// TwinCAT 3 PLC project Press
// ProgramVersion: 3.1.4024.0
// libraries:
//   Tc2_MC2, * (Beckhoff Automation GmbH)
//   Tc2_MC2_Drive, * (Beckhoff Automation GmbH)
//   Tc2_MC2_FlyingSaw, * (Beckhoff Automation GmbH)
//   Tc2_Standard, * (Beckhoff Automation GmbH)
//   Tc2_System, * (Beckhoff Automation GmbH)
//   Tc2_Utilities, * (Beckhoff Automation GmbH)
//   Tc3_Module, * (Beckhoff Automation GmbH)
// project tree:
//   DUTs/ ST_VisionData.TcDUT
//   GVLs/ GVL_Alarm.TcGVL, GVL_Axis01.TcGVL, GVL_Axis02.TcGVL, GVL_Axis03.TcGVL, GVL_Axis04.TcGVL, GVL_Calibration.TcGVL, GVL_Conv.TcGVL, GVL_Encoder.TcGVL, GVL_HMI.TcGVL, GVL_Main_Step.TcGVL, GVL_Mastering.TcGVL, GVL_Motion_Step.TcGVL, GVL_System.TcGVL, GVL_Vision.TcGVL, GVL_Vision_Step.TcGVL
//   / PlcTask.TcTTO
//   POUs/Alarm/ Alarm_Error.TcPOU, Alarm_Warring.TcPOU
//   POUs/Axis01_R/ Axis01_Alarm.TcPOU, Axis01_Auto.TcPOU, Axis01_Command.TcPOU, Axis01_Interlock_ST.TcPOU, Axis01_Manual.TcPOU, Axis01_Status.TcPOU
//   POUs/Axis02_X/ Axis02_Alarm.TcPOU, Axis02_Auto.TcPOU, Axis02_Command.TcPOU, Axis02_Interlock_ST.TcPOU, Axis02_Manual.TcPOU, Axis02_Status.TcPOU
//   POUs/Axis03_Y/ Axis03_Alarm.TcPOU, Axis03_Auto.TcPOU, Axis03_Command.TcPOU, Axis03_Interlock_ST.TcPOU, Axis03_Manual.TcPOU, Axis03_Status.TcPOU
//   POUs/Axis04_Z/ Axis04_Alarm.TcPOU, Axis04_Auto.TcPOU, Axis04_Command.TcPOU, Axis04_Manual.TcPOU, Axis04_Set_Work_End_Speed.TcPOU, Axis04_Status.TcPOU
//   POUs/Axis05_Encoder/ Axis05_Status.TcPOU
//   POUs/ Conv.TcPOU, FB_HomeBeforeMoveAX8000.TcPOU, FB_CamTrigger.TcPOU, FB_LRealRingQueue.TcPOU, FB_VisionDataQueue.TcPOU, MAIN.TcPOU
//   POUs/System/ HMI.TcPOU, HOME_MOVE.TcPOU, Initial.TcPOU, Login_Timer.TcPOU, System.TcPOU
//   POUs/Vision/ Mastering.TcPOU, Move_Command.TcPOU, Vision_ST.TcPOU
//   POUs/Work/ GOST.TcPOU, Motion_Step_ST.TcPOU

CONFIGURATION Press
    RESOURCE PLC ON TwinCAT3
        TASK PlcTask(INTERVAL := T#1ms, PRIORITY := 1);
        PROGRAM MAIN WITH PlcTask : MAIN;
    END_RESOURCE
END_CONFIGURATION

// ---- DUTs/ST_VisionData.TcDUT
(* 비전 결과 1세트 — 큐 적재 단위. 좌표 + 해당 캠트리거 위치를 한 묶음으로 보존. *)
TYPE ST_VisionData :
STRUCT
    ID                : DINT;    // 비전 인식 ID (vision이 부여, 압입 추적용)
    X                 : LREAL;   // Data_Read_X
    Y                 : LREAL;   // Data_Read_Y
    Rot               : LREAL;   // Data_Read_R (R 은 IL Set/Reset 예약어라 Rot 사용)
    Cam_Trig_Position : LREAL;   // 이 결과의 캠트리거 시점 엔코더 위치(Target X 보정 기준)
END_STRUCT
END_TYPE

// ---- GVLs/GVL_Alarm.TcGVL
{attribute 'qualified_only'}
VAR_GLOBAL
	
 	System_Estop_OK			: BOOL 	;
//E-StopAlarm 장비 정지	
	E_STOP_Total_Alarm		: BOOL	;
	E_STOP_Alarm01			: BOOL	;		//EMO-Switch ON
	E_STOP_Alarm02			: BOOL	;		//Door Open
	E_STOP_Alarm03			: BOOL	;		//가이드 축 알람			
	E_STOP_Alarm04			: BOOL	;		//X 축 인터락 알람
	E_STOP_Alarm05			: BOOL	;		//Y 축 인터락 알람
	E_STOP_Alarm06			: BOOL	;		//Z 축 인터락 알람
	E_STOP_Alarm07			: BOOL	;		//R 축 인터락 알람
	E_STOP_Alarm08			: BOOL	;		//비전 RUN OFF 알람
	E_STOP_Alarm09			: BOOL	;
	E_STOP_Alarm10			: BOOL	;		//Vision 통신 이상
	E_STOP_Alarm11			: BOOL	;
	E_STOP_Alarm12			: BOOL	;
	E_STOP_Alarm13			: BOOL	;
	E_STOP_Alarm14			: BOOL	;
	E_STOP_Alarm15			: BOOL	;
	E_STOP_Alarm16			: BOOL	;
	E_STOP_Alarm17			: BOOL	;
	E_STOP_Alarm18			: BOOL	;
	E_STOP_Alarm19			: BOOL	;
	E_STOP_Alarm20			: BOOL	;
//Display Alarm 알람
	Display_Alarm01			: BOOL	;		
	Display_Alarm02			: BOOL	;
	Display_Alarm03			: BOOL	;
	Display_Alarm04			: BOOL	;
	Display_Alarm05			: BOOL	;
	Display_Alarm06			: BOOL	;
	Display_Alarm07			: BOOL	;
	Display_Alarm08			: BOOL	;
	Display_Alarm09			: BOOL	;
	Display_Alarm10			: BOOL	;		//Vision 측정 NG
	Display_Alarm11			: BOOL	;
	Display_Alarm12			: BOOL	;
	Display_Alarm13			: BOOL	;
	Display_Alarm14			: BOOL	;	
	Display_Alarm15			: BOOL	;
//Axis01 Motor Alarm
	Axis01_Total_Alarm		: BOOL	;		
	Axis01_Alarm01			: BOOL	;		
	Axis01_Alarm02			: BOOL	;
	Axis01_Alarm03			: BOOL	;		
	Axis01_Alarm04			: BOOL	;		
	Axis01_Alarm05			: BOOL	;		
	Axis01_Alarm06			: BOOL	;		
	Axis01_Alarm07			: BOOL	;		
	Axis01_Alarm08			: BOOL	;		
	Axis01_Alarm09			: BOOL	;		
	Axis01_Alarm10			: BOOL	;	
	Axis01_Alarm11			: BOOL	;
	Axis01_Alarm12			: BOOL	;			
//Axis02 Motor Alarm
	Axis02_Total_Alarm		: BOOL	;		
	Axis02_Alarm01			: BOOL	;		
	Axis02_Alarm02			: BOOL	;
	Axis02_Alarm03			: BOOL	;		
	Axis02_Alarm04			: BOOL	;		
	Axis02_Alarm05			: BOOL	;		
	Axis02_Alarm06			: BOOL	;		
	Axis02_Alarm07			: BOOL	;		
	Axis02_Alarm08			: BOOL	;		
	Axis02_Alarm09			: BOOL	;		
	Axis02_Alarm10			: BOOL	;
	Axis02_Alarm11			: BOOL	;
	Axis02_Alarm12			: BOOL	;		
//Axis03 Motor Alarm
	Axis03_Total_Alarm		: BOOL	;		
	Axis03_Alarm01			: BOOL	;		
	Axis03_Alarm02			: BOOL	;
	Axis03_Alarm03			: BOOL	;		
	Axis03_Alarm04			: BOOL	;		
	Axis03_Alarm05			: BOOL	;		
	Axis03_Alarm06			: BOOL	;		
	Axis03_Alarm07			: BOOL	;		
	Axis03_Alarm08			: BOOL	;		
	Axis03_Alarm09			: BOOL	;		
	Axis03_Alarm10			: BOOL	;		
	Axis03_Alarm11			: BOOL	;
	Axis03_Alarm12			: BOOL	;
//Axis04 Motor Alarm
	Axis04_Total_Alarm		: BOOL	;		
	Axis04_Alarm01			: BOOL	;		
	Axis04_Alarm02			: BOOL	;
	Axis04_Alarm03			: BOOL	;		
	Axis04_Alarm04			: BOOL	;		
	Axis04_Alarm05			: BOOL	;		
	Axis04_Alarm06			: BOOL	;		
	Axis04_Alarm07			: BOOL	;		
	Axis04_Alarm08			: BOOL	;		
	Axis04_Alarm09			: BOOL	;		
	Axis04_Alarm10			: BOOL	;		
	Axis04_Alarm11			: BOOL	;
	Axis04_Alarm12			: BOOL	;
END_VAR

// ---- GVLs/GVL_Axis01.TcGVL
{attribute 'qualified_only'}
VAR_GLOBAL
//Motor_Status								
    Real_Position						:	LREAL	;		// 실제 위치					
    Real_Velocity						:	LREAL	;		// 실제 속도					
	Busy	   						 	:	BOOL	;		// 동작중			
    Homed       					    :	BOOL	;		// 홈 완료 여부						
    Error								:	BOOL	;		// 에러 발생 여부						
    ErrorID								:	UDINT	;		// 에러 코드						
	StandStill							:	BOOL	;		// 동작가능(축정지,작업명령없음,알람없음)	
	Error_Stop							:	BOOL	;		// 에러 스탑(MC_Reset으로만 해제 가능)
	Power_ON							:	BOOL	;			
	Stop								:	BOOL	;
	Ready								:	BOOL	;		//	모터 Ready
	Home_OK								:	BOOL	;		//	모터 홈 동작 완료
		
//Interlock
	Interlock							:	BOOL	:=	FALSE	;
//Motor_Bit		
	Moving_Command						:	BOOL	;
//Motor_Manual
	M_Home_ORG							:	BOOL	;
	M_Home_Pos_Move						:	BOOL	;
	M_Wait_Pos_Move						:	BOOL	;
	M_Target_Pos_Move					:	BOOL	;
	M_Work_End_Pos_Move					:	BOOL	;
	M_Maint_Pos_Move					:	BOOL	;
	M_Tool_Change_Pos_Move				:	BOOL	;
	M_Calibration_Pos_Move				:	BOOL	;
//Motor_Auto
	A_Home_Pos_Move						:	BOOL	;
	A_Wait_Pos_Move						:	BOOL	;
	A_Target_Pos_Move					:	BOOL	;
	A_Work_End_Pos_Move					:	BOOL	;
	A_Maint_Pos_Move					:	BOOL	;
	A_Tool_Change_Pos_Move				:	BOOL	;
	A_Calibration_Pos_Move				:	BOOL	;
	
//Interlock
	Home_ORG_Interlock					:	BOOL	;
	Home_Pos_Interlock					:	BOOL	;
	Wait_Pos_Interlock					:	BOOL	;
	Target_Pos_Interlock				:	BOOL	;
	Work_End_Pos_Interlock				:	BOOL	;
	Maint_Pos_Interlock					:	BOOL	;
	Tool_Change_Pos_Interlock			:	BOOL	;
	Calibration_Pos_Interlock			:	BOOL	;	
	
	
//Motor_Sensor								
	Home_Sensor  		AT%I*	 		:	 BOOL	;				
	CW_Sensor   		AT%I*			:	 BOOL	;		//Motor +Limit		
	CCW_Sensor  		AT%I*			:	 BOOL	;		//Motor -Limit	
		
//Motor_Position								
	Home_Position						:   BOOL	;						
	Wait_Position						:   BOOL	;						
	Target_Position						:   BOOL	;											
	Work_End_Position					:   BOOL	;
	Maint_Position						:	BOOL	;
	Tool_Change_Position				:	BOOL	;
	Calibration_Position				:	BOOL	;		

//HMI
	HMI_Home_PB							:	BOOL	;
	HMI_Home_Pos_Move_PB				:	BOOL	;
	HMI_Wait_Pos_Move_PB				:	BOOL	;
	HMI_Target_Pos_Move_PB				:	BOOL	;
	HMI_Work_End_Pos_Move_PB			:	BOOL	;
	HMI_Maint_Pos_Move_PB				:	BOOL	;
	HMI_Tool_Change_Move_PB				:	BOOL	;
	HMI_Calibration_Move_PB				:	BOOL	;
	Jog_Forward_PB						:	BOOL	;
	Jog_Backward_PB						:	BOOL	;
	Stop_PB								:	BOOL	;
// Digital Input // P Limit, N Limit
	Digital_Input AT%I*					:	UDINT	;
	
Maint_Position_Data: LREAL;	Power_ON_Delay: BOOL;
	Test_Power_ON: BOOL;
END_VAR
VAR_GLOBAL PERSISTENT
//Motor_Position_Data								
	Home_Position_Data					: 	LREAL	;					
	Wait_Position_Data					: 	LREAL	;					
	Target_Position_Data				: 	LREAL	;							
	Work_End_Position_Data				:	LREAL	;	
	
	Tool_Change_Position_Data			:	LREAL	;
	Calibration_Position_Data			:	LREAL	;
//Motor_Speed_Data
	Work_Speed							:	LREAL	;
	Jog_Speed							:	LREAL	;

END_VAR

VAR_GLOBAL CONSTANT
	Tool_Change_Speed					: 	LREAL := 20 ;
	Calibration_Speed					:	LREAL := 20	;
END_VAR

// ---- GVLs/GVL_Axis02.TcGVL
{attribute 'qualified_only'}
VAR_GLOBAL
//Motor_Status								
    Real_Position						:	LREAL	;		// 실제 위치					
    Real_Velocity						:	LREAL	;		// 실제 속도					
	Busy	   						 	:	BOOL	;		// 동작중			
    Homed       					    :	BOOL	;		// 홈 완료 여부						
    Error								:	BOOL	;		// 에러 발생 여부						
    ErrorID								:	UDINT	;		// 에러 코드						
	StandStill							:	BOOL	;		// 동작가능(축정지,작업명령없음,알람없음)	
	Error_Stop							:	BOOL	;		// 에러 스탑(MC_Reset으로만 해제 가능)
	Power_ON							:	BOOL	;			
	Stop								:	BOOL	;
	Ready								:	BOOL	;		//	모터 Ready
	Home_OK								:	BOOL	;		//	모터 홈 동작 완료
	Work_Offset							:	LREAL	;
	Work_Offset_Move					:	BOOL	;
	Offset_Acceleration					:	LREAL	;
	Accel_Offset						:	LREAL	;
	Speed_Offset						:	LREAL	;
//Interlock
	Interlock							:	BOOL	:=	FALSE	;
//Motor_Bit
	Moving_Command						:	BOOL	;
//Motor_Manual
	M_Home_ORG							:	BOOL	;
	M_Home_Pos_Move						:	BOOL	;
	M_Wait_Pos_Move						:	BOOL	;
	M_Target_Pos_Move					:	BOOL	;
	M_Work_End_Pos_Move					:	BOOL	;
	M_Maint_Pos_Move					:	BOOL	;
	M_Tool_Change_Pos_Move				:	BOOL	;
	M_Calibration_Pos_Move				:	BOOL	;
//Motor_Auto
	A_Home_Pos_Move						:	BOOL	;
	A_Wait_Pos_Move						:	BOOL	;
	A_Target_Pos_Move					:	BOOL	;
	A_Work_End_Pos_Move					:	BOOL	;
	A_Maint_Pos_Move					:	BOOL	;
	A_Tool_Change_Pos_Move				:	BOOL	;
	A_Calibration_Pos_Move				:	BOOL	;
//Interlock
	Home_ORG_Interlock					:	BOOL	;
	Home_Pos_Interlock					:	BOOL	;
	Wait_Pos_Interlock					:	BOOL	;
	Target_Pos_Interlock				:	BOOL	;
	Work_End_Pos_Interlock				:	BOOL	;
	Maint_Pos_Interlock					:	BOOL	;
	Tool_Change_Pos_Interlock			:	BOOL	;
	Calibration_Pos_Interlock			:	BOOL	;
//Motor_Sensor								
	Home_Sensor  		AT%I*	 		:	BOOL	;				
	CW_Sensor   		AT%I*			:	BOOL	;		//Motor +Limit		
	CCW_Sensor  		AT%I*			:	BOOL	;		//Motor -Limit	
		
//Motor_Position								
	Home_Position						:   BOOL	;						
	Wait_Position						:   BOOL	;						
	Target_Position						:   BOOL	;											
	Work_End_Position					:   BOOL	;
	Maint_Position						:	BOOL	;
	Tool_Change_Position				: 	BOOL	;			
	Calibration_Position				: 	BOOL 	;
//HMI
	HMI_Home_PB							:	BOOL	;
	HMI_Home_Pos_Move_PB				:	BOOL	;
	HMI_Wait_Pos_Move_PB				:	BOOL	;
	HMI_Target_Pos_Move_PB				:	BOOL	;
	HMI_Work_End_Pos_Move_PB			:	BOOL	;
	HMI_Maint_Pos_Move_PB				:	BOOL	;
	HMI_Tool_Change_Pos_Move_PB			:	BOOL	;
	HMI_Calibration_Pos_Move_PB			:	BOOL	;
	Jog_Forward_PB						:	BOOL	;
	Jog_Backward_PB						:	BOOL	;
	Stop_PB								:	BOOL	;
//Work_Comp	
	Work_End_Comp						:	BOOL	;
	Home_Comp							:	BOOL	;
// Digital Input // P Limit, N Limit
	Digital_Input AT%I*					: 	UDINT	;




	Power_ON_Delay: BOOL;
	Test_Power_ON: BOOL;
	
END_VAR
VAR_GLOBAL PERSISTENT
//Motor_Position_Data								
	Home_Position_Data					: 	LREAL	;					
	Wait_Position_Data					: 	LREAL	;					
	Target_Position_Data				: 	LREAL	;							
	Work_End_Position_Data				:	LREAL	;
	Maint_Position_Data					:	LREAL	;
	Tool_Change_Position_Data			:	LREAL	;
	Calibration_Position_Data			:	LREAL	;
//Motor_Speed_Data
	Work_Speed							:	LREAL	;
	

END_VAR

VAR_GLOBAL CONSTANT
	Tool_Change_Speed					: 	LREAL := 20 ;
	Calibration_Speed					:	LREAL := 20	;
	Sync_Data							:	LREAL := 20 ;
	Jog_Speed							:	LREAL := 20	;
END_VAR

// ---- GVLs/GVL_Axis03.TcGVL
{attribute 'qualified_only'}
VAR_GLOBAL
//Motor_Status								
    Real_Position						:	LREAL	;		// 실제 위치					
    Real_Velocity						:	LREAL	;		// 실제 속도					
	Busy	   						 	:	BOOL	;		// 동작중			
    Homed       					    :	BOOL	;		// 홈 완료 여부						
    Error								:	BOOL	;		// 에러 발생 여부						
    ErrorID								:	UDINT	;		// 에러 코드						
	StandStill							:	BOOL	;		// 동작가능(축정지,작업명령없음,알람없음)	
	Error_Stop							:	BOOL	;		// 에러 스탑(MC_Reset으로만 해제 가능)
	Power_ON							:	BOOL	;			
	Stop								:	BOOL	;
	Ready								:	BOOL	;		//	모터 Ready
	Home_OK								:	BOOL	;		//	모터 홈 동작 완료

//Interlock
	Interlock							:	BOOL	:=	FALSE	;
//Motor_Bit
	Moving_Command						:	BOOL	;
//Motor_Manual
	M_Home_ORG							:	BOOL	;
	M_Home_Pos_Move						:	BOOL	;
	M_Wait_Pos_Move						:	BOOL	;
	M_Target_Pos_Move					:	BOOL	;
	M_Work_End_Pos_Move					:	BOOL	;
	M_Maint_Pos_Move					:	BOOL	;
	M_Tool_Change_Pos_Move				:	BOOL	;
	M_Calibration_Pos_Move				:	BOOL	;
//Motor_Auto
	A_Home_Pos_Move						:	BOOL	;
	A_Wait_Pos_Move						:	BOOL	;
	A_Target_Pos_Move					:	BOOL	;
	A_Work_End_Pos_Move					:	BOOL	;
	A_Maint_Pos_Move					:	BOOL	;
	A_Tool_Change_Pos_Move				:	BOOL	;
	A_Calibration_Pos_Move				:	BOOL	;
//Interlock
	Home_ORG_Interlock					:	BOOL	;
	Home_Pos_Interlock					:	BOOL	;
	Wait_Pos_Interlock					:	BOOL	;
	Target_Pos_Interlock				:	BOOL	;
	Work_End_Pos_Interlock				:	BOOL	;
	Maint_Pos_Interlock					:	BOOL	;
	Tool_Change_Pos_Interlock			:	BOOL	;
	Calibration_Pos_Interlock			:	BOOL	;

	
//Motor_Sensor								
	Home_Sensor  		AT%I*	 		:	 BOOL	;				
	CW_Sensor   		AT%I*			:	 BOOL	;		//Motor +Limit		
	CCW_Sensor  		AT%I*			:	 BOOL	;		//Motor -Limit	
	
//Motor_Position								
	Home_Position						:   BOOL	;						
	Wait_Position						:   BOOL	;						
	Target_Position						:   BOOL	;											
	Work_End_Position					:   BOOL	;
	Maint_Position						:	BOOL	;
	Tool_Change_Position				:	BOOL	;	
	Calibration_Position				: 	BOOL	;
//HMI
	HMI_Home_PB							:	BOOL	;
	HMI_Home_Pos_Move_PB				:	BOOL	;
	HMI_Wait_Pos_Move_PB				:	BOOL	;
	HMI_Target_Pos_Move_PB				:	BOOL	;
	HMI_Work_End_Pos_Move_PB			:	BOOL	;
	HMI_Maint_Pos_Move_PB				:	BOOL	;
	HMI_Tool_Change_Pos_Move_PB			:	BOOL	;
	HMI_Calibration_Pos_Move_PB			:	BOOL	;
	Jog_Forward_PB						:	BOOL	;
	Jog_Backward_PB						:	BOOL	;
	Stop_PB								:	BOOL	;
	
// Digital Input // P Limit, N Limit
	Digital_Input AT%I*					:	UDINT	;

	Power_ON_Delay: BOOL;
	Test_Power_ON: BOOL;
END_VAR
VAR_GLOBAL PERSISTENT
//Motor_Position_Data								
	Home_Position_Data					: 	LREAL	;					
	Wait_Position_Data					: 	LREAL	;					
	Target_Position_Data				: 	LREAL	;							
	Work_End_Position_Data				:	LREAL	;		
	Maint_Position_Data					:	LREAL	;
	Tool_Change_Position_Data			:	LREAL	;
	Calibration_Position_Data			:	LREAL	;
//Motor_Speed_Data
	Work_Speed							:	LREAL	;
	Jog_Speed							:	LREAL	;
	
END_VAR

VAR_GLOBAL CONSTANT
	Calibration_Speed					: 	LREAL	:= 20;
	Tool_Change_Speed					: 	LREAL	:= 20;
END_VAR

// ---- GVLs/GVL_Axis04.TcGVL
{attribute 'qualified_only'}
VAR_GLOBAL
//Motor_Status								
    Real_Position						:	LREAL	;		// 실제 위치					
    Real_Velocity						:	LREAL	;		// 실제 속도					
	Busy	   						 	:	BOOL	;		// 동작중			
    Homed       					    :	BOOL	;		// 홈 완료 여부						
    Error								:	BOOL	;		// 에러 발생 여부						
    ErrorID								:	UDINT	;		// 에러 코드						
	StandStill							:	BOOL	;		// 동작가능(축정지,작업명령없음,알람없음)	
	Error_Stop							:	BOOL	;		// 에러 스탑(MC_Reset으로만 해제 가능)
	Power_ON							:	BOOL	;			
	Stop								:	BOOL	;
	Ready								:	BOOL	;		//	모터 Ready
	Home_OK								:	BOOL	;		//	모터 홈 동작 완료
	
//Interlock
	Interlock							:	BOOL	:=	FALSE	;
//Motor_Bit
	Moving_Command						:	BOOL	;
M_Home_ORG: BOOL;
	M_Home_Pos_Move						:	BOOL	;
	M_Wait_Pos_Move						:	BOOL	;
	M_Target_Pos_Move					:	BOOL	;
	M_Work_End_Pos_Move					:	BOOL	;
	M_Maint_Pos_Move					:	BOOL	;
	M_Tool_Change_Pos_Move				:	BOOL	;
	M_Calibration_Pos_Move				:	BOOL	;
//Motor_Auto
	A_Home_Pos_Move						:	BOOL	;
	A_Wait_Pos_Move						:	BOOL	;
	A_Target_Pos_Move					:	BOOL	;
	A_Work_End_Pos_Move					:	BOOL	;
	A_Maint_Pos_Move					:	BOOL	;
	A_Tool_Change_Pos_Move				:	BOOL	;
	A_Calibration_Pos_Move				:	BOOL	;
//Interlock
	Home_ORG_Interlock					:	BOOL	;
	Home_Pos_Interlock					:	BOOL	;
	Wait_Pos_Interlock					:	BOOL	;
	Target_Pos_Interlock				:	BOOL	;
	Work_End_Pos_Interlock				:	BOOL	;
	Maint_Pos_Interlock					:	BOOL	;
	Tool_Change_Pos_Interlock			:	BOOL	;
	Calibration_Pos_Interlock			:	BOOL	;
	
//Motor_Sensor								
	Home_Sensor  		AT%I*		 	:	 BOOL	;				
	CW_Sensor   		AT%I*			:	 BOOL	;		//Motor +Limit		
	CCW_Sensor  		AT%I*			:	 BOOL	;		//Motor -Limit	
		
//Motor_Position								
	Home_Position						:   BOOL	;						
	Wait_Position						:   BOOL	;						
	Target_Position						:   BOOL	;											
	Work_End_Position					:   BOOL	;
	Maint_Position						:	BOOL	;
	Tool_Change_Position				:	BOOL	;
	Calibration_Position				:	BOOL	;			

//HMI
	HMI_Home_PB							:	BOOL	;
	HMI_Home_Pos_Move_PB				:	BOOL	;
	HMI_Wait_Pos_Move_PB				:	BOOL	;
	HMI_Target_Pos_Move_PB				:	BOOL	;
	HMI_Work_End_Pos_Move_PB			:	BOOL	;
	HMI_Maint_Pos_Move_PB				:	BOOL	;
	HMI_Tool_Change_Pos_Move_PB			:	BOOL	;
	HMI_Calibration_Pos_Move_PB			:	BOOL	;
	Jog_Forward_PB						:	BOOL	;
	Jog_Backward_PB						:	BOOL	;
	Stop_PB								:	BOOL	;	

// Digital Input // P Limit, N Limit
	Digital_Input AT%I*					: 	UDINT	;	


	Power_ON_Delay: BOOL;
	Test_Power_ON: BOOL;
	
	M_Cleaning_Move: BOOL;
	Cleaning_Move_Position: BOOL;
	M_Mastering_Pos_Move: BOOL;
	Mastering_Position: BOOL;
END_VAR
VAR_GLOBAL PERSISTENT
//Motor_Position_Data								
	Home_Position_Data					: 	LREAL	;					
	Wait_Position_Data					: 	LREAL	;					
	Target_Position_Data				: 	LREAL	;							
	Work_End_Position_Data				:	LREAL	;	
	Maint_Position_Data					:	LREAL	;
	Tool_Change_Position_Data			:	LREAL	;
	Calibration_Position_Data			:	LREAL	;	
	Cleaning_Move_Data: LREAL := 0;
//Motor_Speed_Data
	Work_Speed							:	LREAL	;
	Jog_Speed							:	LREAL	;

//Motor_Torque_Data
	Torque_UP_Limit				AT%Q*	:	UINT	;
	Torque_Down_Limit			AT%Q*	:	UINT	;
	Wait_Speed							: 	LREAL	;
END_VAR

VAR_GLOBAL CONSTANT
	Calibration_Speed					: 	LREAL	:= 20;
	Tool_Change_Speed					: 	LREAL	:= 20;
END_VAR

// ---- GVLs/GVL_Calibration.TcGVL
{attribute 'qualified_only'}
VAR_GLOBAL
	Calibration_Pos_Moving			: 	BOOL	;
	HMI_Calibration_Pos_Move_PB		: 	BOOL	;
	Calibration_comp				: 	BOOL	;
	Calibration_OK					: 	BOOL	;
	All_Motor_Wait_Pos_Moving		: 	BOOL	;
	Calibration_Pos_Interlock 		: 	BOOL	;
	Data_Read_Comp					: 	BOOL	;
	Axis01_Data_Apply_Comp			: 	BOOL	;
	Axis02_Data_Apply_Comp			: 	BOOL	;
	Axis03_Data_Apply_Comp			: 	BOOL	;
	Axis04_Data_Apply_Comp			:   BOOL;
	Motor_Move : BOOL := FALSE;
	
END_VAR

// ---- GVLs/GVL_Conv.TcGVL
{attribute 'qualified_only'}
VAR_GLOBAL
	
	Auto_Mode					AT%I*	:	BOOL	;	// 컨베이어 자동 스위치
	E_STOP						AT%I*	:	BOOL	;	// 컨베이어 E_STOP


	//Output Card 01
	Conv_Motor_CW				AT%Q*	:	BOOL	;	// 컨베이어 전진
	Conv_Motor_CCW				AT%Q*	:	BOOL	;	// 컨베이어 후진
	Conv_Motor_High_Speed		AT%Q*	:	BOOL	;	// 컨베이어 고속
	Conv_Motor_Normal_Speed		AT%Q*	:	BOOL	;	// 컨베이어 중속
	Conv_Motor_Low_Speed		AT%Q*	:	BOOL	;	// 컨베이어 저속

	HMI_Motor_CW						:	BOOL	;	// HMI 컨베이어 전진
	HMI_Motor_CCW						:	BOOL	;	// HMI 컨베이어 후진 
	HMI_Motor_High_Speed				:	BOOL	;	// HMI 컨베이어 고속
	HMI_Motor_Normal_Speed				:	BOOL	;	// HMI 컨베이어 중속
	HMI_Motor_Low_Speed					:	BOOL	;	// HMI 컨베이어 저속
	
	Motor_STOP							:	BOOL	;


	

	

END_VAR

// ---- GVLs/GVL_Encoder.TcGVL
{attribute 'qualified_only'}
VAR_GLOBAL
	Enc_Axis: AXIS_REF;
	Conveyor_Speed :	LREAL	;
	Encoder_Value	:	LREAL	;
	Real_Position: LREAL;
	Real_Velocity: LREAL;
	Count	AT%I*	:INT;
	Conveyor_CW AT%Q* : BOOL	;
	Conveyor_CCW AT%Q* : BOOL	;
	
END_VAR

// ---- GVLs/GVL_HMI.TcGVL
{attribute 'qualified_only'}
VAR_GLOBAL

// HMI Screen NO
    NowScreen_NO            :    INT    ;       // 현재 화면 위치 NO
	ChangeScreen_NO         :    INT    ;       // PLC 요구 화면 NO

	
// HMI 화면 전환	
	AXIS01					:	BOOL	;
	AXIS02					:	BOOL	;
	AXIS03					:	BOOL	;
	AXIS04					:	BOOL	;
	
	AXIS01_LAMP				:	BOOL	;
	AXIS02_LAMP				:	BOOL	;
	AXIS03_LAMP				:	BOOL	;
	AXIS04_LAMP				:	BOOL	;
END_VAR

// ---- GVLs/GVL_Main_Step.TcGVL
{attribute 'qualified_only'}
VAR_GLOBAL
	Status						:	BOOL	;
	NO							:	INT		;
	Wait_Vision					: 	BOOL	;
	Data_Copy					:	BOOL	;
	Vision_Data_Apply			: 	BOOL	;
	Wait_Start_Sensor			: 	BOOL	;
	Moving_Start				: 	BOOL	;
	Axis04_Comp					: 	BOOL	;
	Axis04_Work_Comp			: 	BOOL	;
	Axis04_Work_Comp_Wait		: 	BOOL	;
	Press_5ms					: 	BOOL	;
	Press_Stop					:	BOOL	;
	Axis04_Wait_Pos_Moving		: 	BOOL	;
	Axis02_Work_Comp_Wait		: 	BOOL	;
	Axis02_Wait_Pos_Moving		: 	BOOL	;
	All_Motor_Wait_Pos_Moving	:	BOOL	;
	Vision_Data_Reset			:	BOOL	;
	Vision_Data_Initial			:	BOOL	;
	All_Initial					:	BOOL	;
	Target_Position_Moving		:	BOOL	;
	Press_Start					:	BOOL	;
	Press_Wait					:	BOOL	;
	Axis04_Work_move			:	BOOL	;
	

	Data_Copy_Comp				:	BOOL	;
END_VAR

// ---- GVLs/GVL_Mastering.TcGVL
{attribute 'qualified_only'}
VAR_GLOBAL
	Case_Length_Check_Start 	: 	BOOL;
	Case_Length					:	LREAL;
	mastering_vision_x			:	LREAL;
	Back_Shot_Position			:	LREAL;
	Reshot_Position				:	LREAL;
	Back_Trig					: 	BOOL;
END_VAR

// ---- GVLs/GVL_Motion_Step.TcGVL
{attribute 'qualified_only'}
VAR_GLOBAL
	Status: BOOL;
	No: INT;
	Target_Pos_Moving: BOOL;
	Motion_Start: BOOL;
	Axis02_Work_Wait: BOOL;
	Press_Start: BOOL;
	Axis04_Torque_Controll: BOOL;
	Axis04_Wait_Pos_Moving: BOOL;
	All_Axis_Wait_Pos_Moving: BOOL;
	Work_Comp_Target_Pos_Moving: BOOL;
	All_Initial: BOOL;
	Axis02_Stop: BOOL;
	Z_Press_Start: BOOL;
	Force_Gear_Out: BOOL;   // 실패 abort 시 X축 gear-out 강제 (→ Axis02_Command MC_GearOut.Execute OR 입력)
END_VAR

// ---- GVLs/GVL_System.TcGVL
{attribute 'qualified_only'}
VAR_GLOBAL
// Glovel Bit
	Pulse_100ms					:	BOOL	;			//0.1s Bit
	Pulse_1S					:	BOOL	;			//1S Bit		
// System Bit
	Manual_Mode					:	BOOL	;			//HMI 메뉴얼 모드
	Auto_Mode					:	BOOL	;			//HMI 오토모드
	Stop						:	BOOL	;			//HMI Stop
	Safety_ALL_OK				:	BOOL	;			//EMO+Door
	Test_Mode					:	BOOL	;
	All_Initial					:	BOOL	;
	ToggleBit					:	BOOL	;
	Door_Bypass		AT%Q*		:	BOOL	;			//도어 인터록 바이패스 릴레이 출력 (EL2809 Ch11)
//EMO SW	
	EMO_SWitch		AT%I*		:	BOOL	;

//Fiber Sensor
	Fiber_Sensor	AT%I*	:	BOOL	;

//System_Door_Sensor
	Door_Open		AT%I*		:	BOOL	;

//TowerLamp
	Tower_Lamp_Green	AT%Q*	:	BOOL	;
	Tower_Lamp_Yellow	AT%Q*	:	BOOL	;
	Tower_Lamp_Red		AT%Q*	:	BOOL	;
	Buzzer				AT%Q*	:	BOOL	;
//HMI
	Buzzer_Stop						AT%I*	:	BOOL	;
	Alarm_Reset						AT%I*	:	BOOL	;
//Panel
	DC01_SMPS_OK					AT%I*	:	BOOL	;
	DC02_SMPS_OK					AT%I*	:	BOOL	;
	DC03_SMPS_OK					AT%I*	:	BOOL	;
	Servo_Drive_Control_DC_Power	AT%I*	:	BOOL	;
	Inverter_Power_OK					AT%I*	:	BOOL	;
	Inverter_MC_OK					AT%I*	:	BOOL	;
	MC_OK							AT%I*	:	BOOL	;
	CAM_TRIGGER_FAIL				AT%I*	:	BOOL	;
	Main_Lamp_ON					AT%I*	:	BOOL	;
	PC_Power_CP						AT%I*	:	BOOL	;
	CAM_Lamp_CP						AT%I*	:	BOOL	;
	Ps01_Power_OK					AT%I*	:	BOOL	;
	HMI_Power_OK					AT%I*	:	BOOL	;
	Cam_Power_OK					AT%I*	:	BOOL	;
	Inverter_Alarm_ON					AT%I*	:	BOOL	;
	
	
//Bool
	HMI_Auto_Mode				:	BOOL	;		//HMI 오토모드
	ALL_Motor_Homed				:	BOOL	;		//전체 모터 홈 OK
	ALL_Motor_Home_Position		:	BOOL	;		//전체 모터 홈포지션
	HMI_Manual_Mode				:	BOOL	;		//HMI 메뉴얼 모드
	ALL_Motor_Busy				:	BOOL	;		//전체 모터 동작중
	ALL_Motor_StandStill		:	BOOL	;		//전체 모터 동작 가능
	Moving_Motor_Wait_Position	:	BOOL	;		//X,Y,Z,R Wait Position
	Each_Motor_Homed			:	BOOL	;		//개별 로못 홈
	Each_Motor_Busy				:	BOOL	;		//개별 로봇 동작중
	All_Motor_Stop				:	BOOL	;	
	
	
	
	Test_Data_Read_Comp			: 	BOOL	;
	Test_Continues				: 	BOOL	;
	Calibration_Mode			: 	BOOL	;
	Tool_Change_Mode			: 	BOOL	;
	Tool_Change_Move_PB			: 	BOOL	;	
//홈동작 
	ALL_Wait_Position			: 	BOOL	;
	ALL_Home_Move_PB			:	BOOL	;
	ALL_Home_Move_Start			:	BOOL	;
	Axis01_Home_Move			: 	BOOL	;
	Axis02_Home_Move			: 	BOOL	;
	Axis03_Home_Move			: 	BOOL	;
	Axis04_Home_Move			: 	BOOL	;
	
	Axis01_Home_Pos_Move		: 	BOOL	;
	Axis04_Wait_Pos_Move		:	BOOL	;
	Axis03_Wait_Pos_Move		: 	BOOL	;
	Axis01_Wait_Pos_Move		: 	BOOL	;
	Axis02_Wait_Pos_Move		: 	BOOL	;
	Calibration_PB				: 	BOOL	;
	Test_Start					: 	BOOL	;
	
//현재 시간
	Time_Data 					: 	ULINT	; 
	
	Offset_Value				:	LREAL	;
	Task_Offset					:	LREAL	;
	Task_Time					:	LREAL	;

	CV_STOP: BOOL;
	

	Manual_Door_Bypass			: 	BOOL	;
	HMI_Door_Bypass				: 	BOOL	;
	Login						: 	BOOL	;
	LoginLamp					:	BOOL	;
	All_Axis_Wait_Pos_Moving: BOOL;
	Add_Case_Mode: BOOL;
	
	GOST_MODE					:	BOOL	;
END_VAR

// ---- GVLs/GVL_Vision.TcGVL
{attribute 'qualified_only'}
VAR_GLOBAL
//Vision_Bool
	Data_Read_Comp							:	BOOL	;
	Data_Read_OK							:	BOOL	;
	Data_Read_NG							:	BOOL	;
	Axis01_Data_Apply_Comp					:	BOOL	;
	Axis02_Data_Apply_Comp					:	BOOL	;
	Axis03_Data_Apply_Comp					:	BOOL	;
	Cam_Trigger					AT%Q*		:	BOOL	;
	Vision_OK								:	BOOL	;
	Vision_Light_ON				AT%Q*		:	BOOL 	;
	Data_Empty								:	BOOL	;

//Vision Data
	Data_Read_ID							:	DINT	;	// 비전 인식 ID (vision이 부여, X/Y/R·Vision_OK 와 함께 전송)
	Data_Read_X								:	LREAL	;
	Data_Read_Y								:	LREAL	;
	Data_Read_R								:	LREAL	;
	Target_X_Real_Position_Data				:	LREAL	;
	ON_Delay_Time							:	LREAL	;
	Start_Pos_Data							:	LREAL	;
	Sensor_Trig_Pos							:	LREAL	;	// fiber 센서 감지 시점 엔코더 위치 (카메라 트리거 기준점)
	Cam_Trig_Position						:	LREAL	;	// 오토모드 카메라 트리거 시점 엔코더 위치 (Target X 보정 기준)

//Vision_Status
	Vision_Alarm_Code						:	INT		;


	Axis01_Calibration_Position_Data_Old	:	LREAL	;
	Axis02_Calibration_Position_Data_Old	:	LREAL	;
	Axis03_Calibration_Position_Data_Old	:	LREAL	;
	Axis04_Calibration_Position_Data_Old	:	LREAL   ;

	Axis02_Tool_Change_Position_Data		:	LREAL	;
	Axis03_Tool_Change_Position_Data		:	LREAL	;
	Axis04_Tool_Change_Position_Data		:	LREAL	;


//Vision_Data_Buffer

	Data_Buffer_X							:	LREAL	;
	Data_Buffer_Y							:	LREAL	;
	Data_Buffer_R							:	LREAL	;


	Data_Check: BOOL;

	Vision_Q_Overflow						:	BOOL	;	// 비전 결과 큐 만재(무음 유실 경보)
	Vision_Q_Count							:	INT		;	// 비전 결과 큐 적재 수(모니터)

//Press 추적 (vision 대시보드용, 무손실 링버퍼) — vision은 각 Count 증가분만큼 Buf[(idx) MOD 256] 읽음
	Pressed_ID_Buf		: ARRAY[0..255] OF DINT;	// 압입된 인식 ID
	Skipped_ID_Buf		: ARRAY[0..255] OF DINT;	// 건너뛴 인식 ID
	Skipped_Reason_Buf	: ARRAY[0..255] OF INT;		// 건너뛴 사유 (1=Wait지나 도달불가폐기, 2=R/Y지연 미압입abort, 3=큐만재 거부)

	Stop_On_Fail		:	BOOL	;	// (vision 이 ON/OFF) TRUE 면 프레스 실패 시 컨베이어 정지 + 수동 전환. 기본 FALSE(안전)


END_VAR
VAR_GLOBAL PERSISTENT
	Cam_Trigger_Length						:	LREAL	;
	Axis04_Mastering_Position_Data: LREAL := -20;
	Press_Count : UDINT;   // 실제 압입(Z 압입완료) 누적 횟수(전원 유지) — Pressed_ID_Buf 읽기 기준
	Skip_Count  : UDINT;   // 건너뛴 누적 횟수(전원 유지) — Skipped_ID/Reason_Buf 읽기 기준
END_VAR

VAR_GLOBAL CONSTANT
	Axis01_Calibration_Position_Data		:	LREAL := -5	;
	Axis02_Calibration_Position_Data		:	LREAL := 80	;
	Axis03_Calibration_Position_Data		:	LREAL := -10	;
	Axis04_Calibration_Position_Data		:	LREAL := -20	;
END_VAR

// ---- GVLs/GVL_Vision_Step.TcGVL
{attribute 'qualified_only'}
VAR_GLOBAL
//INT
	NO					:	INT		;
//Bool
	Status				:	BOOL	;
	Vision_Start		:	BOOL	;
	Wait_Vision_OK		:	BOOL	;
	Data_Copy: BOOL;
	Data_Initial: BOOL;
	Data_Copy_Check: BOOL;
END_VAR

// ---- POUs/MAIN.TcPOU
PROGRAM MAIN
VAR
END_VAR

//Axis01: R
Axis01_Status();
Axis01_Command();
Axis01_Manual();
Axis01_Auto();
Axis01_Alarm();

//Axis02: X
Axis02_Status();
Axis02_Command();
Axis02_Manual();
Axis02_Auto();
Axis02_Alarm();

//Axis03: Y
Axis03_Status();
Axis03_Command();
Axis03_Manual();
Axis03_Auto();
Axis03_Alarm();

//Axis04: Z
Axis04_Status();
Axis04_Command();
Axis04_Manual();
Axis04_Auto();
Axis04_Alarm();

//Axis05: Encoder
Axis05_Status();

Conv();
//Alarm
Alarm_Error();
Alarm_Warring();

//System
HMI();
HOME_MOVE();
Initial();
System();

//Vision
Vision_ST();
Move_Command();

//Work
Motion_Step_ST();

Mastering();

GOST();

END_PROGRAM

// ---- POUs/Axis01_R/Axis01_Status.TcPOU
PROGRAM Axis01_Status
VAR
//System_Bit
	Always_ON	:	BOOL	:=TRUE	;//상시 ON 
	Always_OFF	:	BOOL	:=FALSE	;//상시 OFF
	Axis01_Status_01: MC_ReadStatus;
	Axis01_Position_Read_01: MC_ReadActualPosition;
	Axis01_Velocity_Read_01: MC_ReadActualVelocity;
	Axis01_Reset_01: MC_Reset;
	Axis01_Stop_01: MC_Stop;
END_VAR

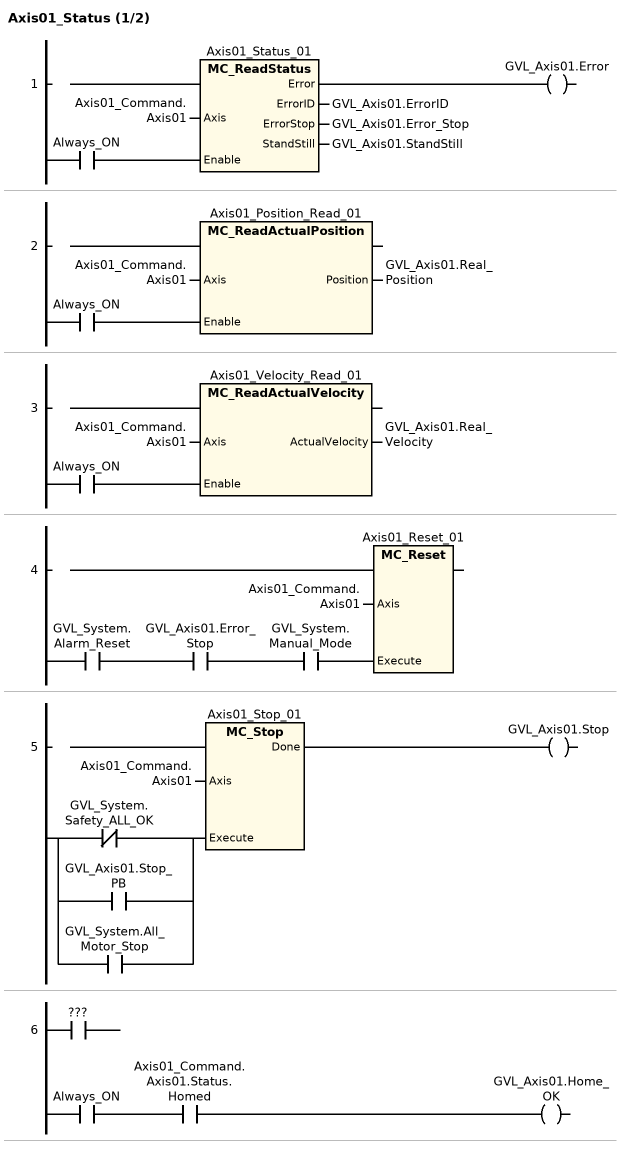
// NETWORK 1
Axis01_Status_01(
    Axis := Axis01_Command.Axis01,
    Enable := Always_ON,
    Error => GVL_Axis01.Error,
    ErrorID => GVL_Axis01.ErrorID,
    ErrorStop => GVL_Axis01.Error_Stop,
    StandStill => GVL_Axis01.StandStill); // MC_ReadStatus

// NETWORK 2
Axis01_Position_Read_01(
    Axis := Axis01_Command.Axis01,
    Enable := Always_ON,
    Position => GVL_Axis01.Real_Position); // MC_ReadActualPosition

// NETWORK 3
Axis01_Velocity_Read_01(
    Axis := Axis01_Command.Axis01,
    Enable := Always_ON,
    ActualVelocity => GVL_Axis01.Real_Velocity); // MC_ReadActualVelocity

// NETWORK 4
Axis01_Reset_01(Axis := Axis01_Command.Axis01, Execute := GVL_System.Alarm_Reset AND GVL_Axis01.Error_Stop AND GVL_System.Manual_Mode); // MC_Reset

// NETWORK 5
Axis01_Stop_01(Axis := Axis01_Command.Axis01, Execute := NOT GVL_System.Safety_ALL_OK OR GVL_Axis01.Stop_PB OR GVL_System.All_Motor_Stop); // MC_Stop
GVL_Axis01.Stop := Axis01_Stop_01.Done;

// NETWORK 6
GVL_Axis01.Home_OK := Always_ON AND Axis01_Command.Axis01.Status.Homed;

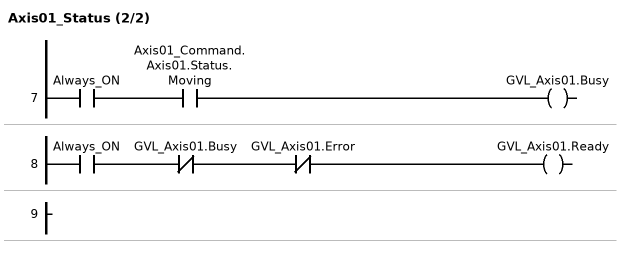
// NETWORK 7
GVL_Axis01.Busy := Always_ON AND Axis01_Command.Axis01.Status.Moving;

// NETWORK 8
GVL_Axis01.Ready := Always_ON AND NOT GVL_Axis01.Busy AND NOT GVL_Axis01.Error;

// NETWORK 9

END_PROGRAM

// ---- POUs/Axis01_R/Axis01_Command.TcPOU
PROGRAM Axis01_Command
VAR
	Axis01: AXIS_REF;											//회전축
	Axis01_MC_Home: FB_HomeBeforeMoveAX8000;
	Axis01_MC_Power: MC_Power;
	Axis01_Status: MC_ReadStatus;
	Axis01_Position_Read: MC_ReadActualPosition;
	Axis01_Velocity_Read: MC_ReadActualVelocity;
	Axis01_Reset: MC_Reset;										//모터 알람 리셋
	Axis01_Stop: MC_Stop;										//모터 정지
	Axis01_Press_Move: MC_MoveAbsolute;
	Axis01_Home_Pos_Move: MC_MoveAbsolute;
	Axis01_Wait_Pos_Move: MC_MoveAbsolute;
	Axis01_Target_Pos_Move: MC_MoveAbsolute;
	Axis01_Work_End_Move: MC_MoveAbsolute;
	Axis01_Jog: MC_Jog;
	
	Always_ON	:	BOOL	:=TRUE	;//상시 ON
	Always_OFF	:	BOOL	:=FALSE	;//상시 OFF

	Home_Interlock			:	BOOL	;
	Home_Pos_Interlock		: 	BOOL	;
	Wait_Pos_Interlock		:	BOOL	;
	Target_Pos_Interlock	:	BOOL	;
	Work_End_POs_Interlock	:	BOOL	;
	Axis01_Calibration: MC_MoveAbsolute;
	Axis01_Maint_Move: MC_MoveAbsolute;
	Axis01_Tool_Change_Move: MC_MoveAbsolute;
	Axis01_Calibration_Move: MC_MoveAbsolute;
	Timer04: TON;
	keb_R: BOOL;
END_VAR
VAR // added by the converter: edge detectors and wires of the graphical bodies
    _rt1 : R_TRIG;
END_VAR

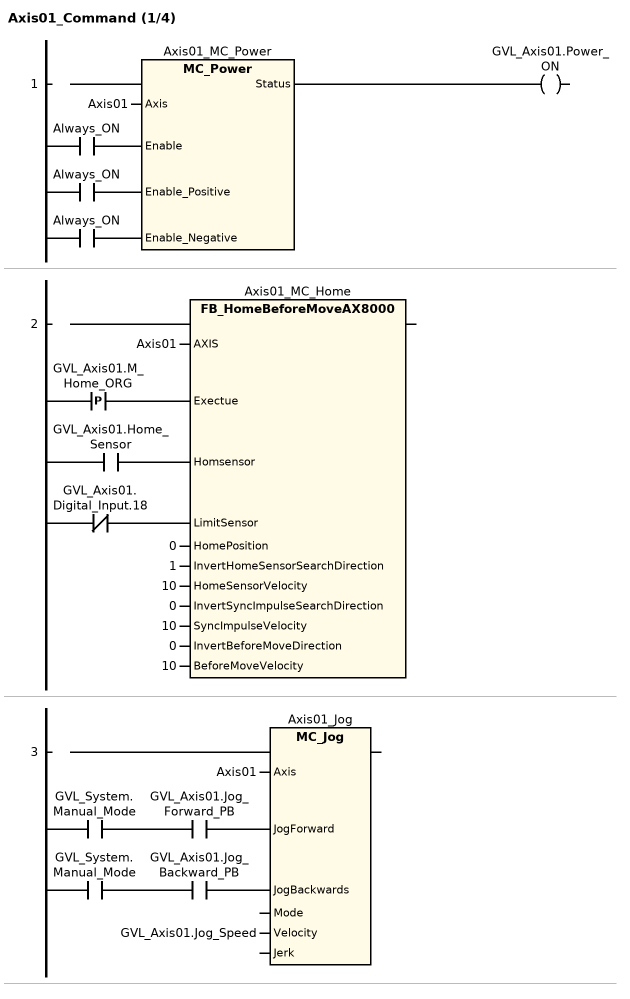
// NETWORK 1
Axis01_MC_Power(
    Axis := Axis01,
    Enable := Always_ON,
    Enable_Positive := Always_ON,
    Enable_Negative := Always_ON); // MC_Power
GVL_Axis01.Power_ON := Axis01_MC_Power.Status;

// NETWORK 2
_rt1(CLK := GVL_Axis01.M_Home_ORG);
Axis01_MC_Home(
    AXIS := Axis01,
    Exectue := _rt1.Q,
    Homsensor := GVL_Axis01.Home_Sensor,
    LimitSensor := NOT GVL_Axis01.Digital_Input.18,
    HomePosition := 0,
    InvertHomeSensorSearchDirection := 1,
    HomeSensorVelocity := 10,
    InvertSyncImpulseSearchDirection := 0,
    SyncImpulseVelocity := 10,
    InvertBeforeMoveDirection := 0,
    BeforeMoveVelocity := 10); // FB_HomeBeforeMoveAX8000

// NETWORK 3
Axis01_Jog(
    Axis := Axis01,
    JogForward := GVL_System.Manual_Mode AND GVL_Axis01.Jog_Forward_PB,
    JogBackwards := GVL_System.Manual_Mode AND GVL_Axis01.Jog_Backward_PB,
    Velocity := GVL_Axis01.Jog_Speed); // MC_Jog

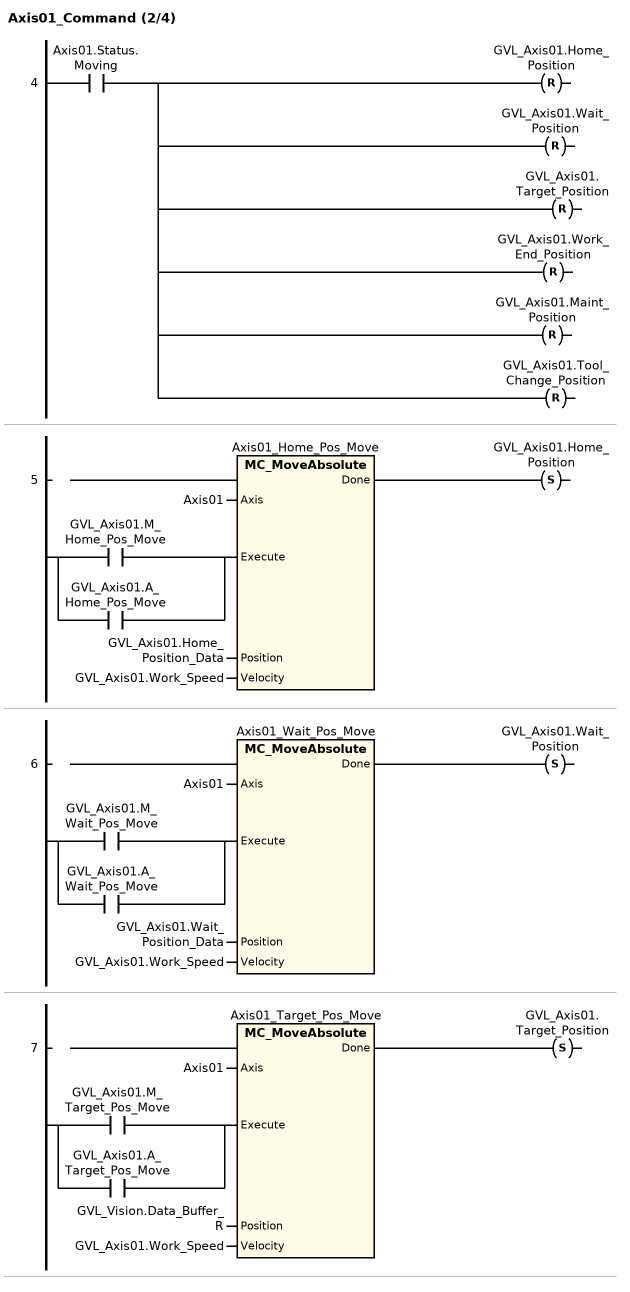
// NETWORK 4
GVL_Axis01.Home_Position R= Axis01.Status.Moving;
GVL_Axis01.Wait_Position R= Axis01.Status.Moving;
GVL_Axis01.Target_Position R= Axis01.Status.Moving;
GVL_Axis01.Work_End_Position R= Axis01.Status.Moving;
GVL_Axis01.Maint_Position R= Axis01.Status.Moving;
GVL_Axis01.Tool_Change_Position R= Axis01.Status.Moving;

// NETWORK 5
Axis01_Home_Pos_Move(
    Axis := Axis01,
    Execute := GVL_Axis01.M_Home_Pos_Move OR GVL_Axis01.A_Home_Pos_Move,
    Position := GVL_Axis01.Home_Position_Data,
    Velocity := GVL_Axis01.Work_Speed); // MC_MoveAbsolute
GVL_Axis01.Home_Position S= Axis01_Home_Pos_Move.Done;

// NETWORK 6
Axis01_Wait_Pos_Move(
    Axis := Axis01,
    Execute := GVL_Axis01.M_Wait_Pos_Move OR GVL_Axis01.A_Wait_Pos_Move,
    Position := GVL_Axis01.Wait_Position_Data,
    Velocity := GVL_Axis01.Work_Speed); // MC_MoveAbsolute
GVL_Axis01.Wait_Position S= Axis01_Wait_Pos_Move.Done;

// NETWORK 7
Axis01_Target_Pos_Move(
    Axis := Axis01,
    Execute := GVL_Axis01.M_Target_Pos_Move OR GVL_Axis01.A_Target_Pos_Move,
    Position := GVL_Vision.Data_Buffer_R,
    Velocity := GVL_Axis01.Work_Speed); // MC_MoveAbsolute
GVL_Axis01.Target_Position S= Axis01_Target_Pos_Move.Done;

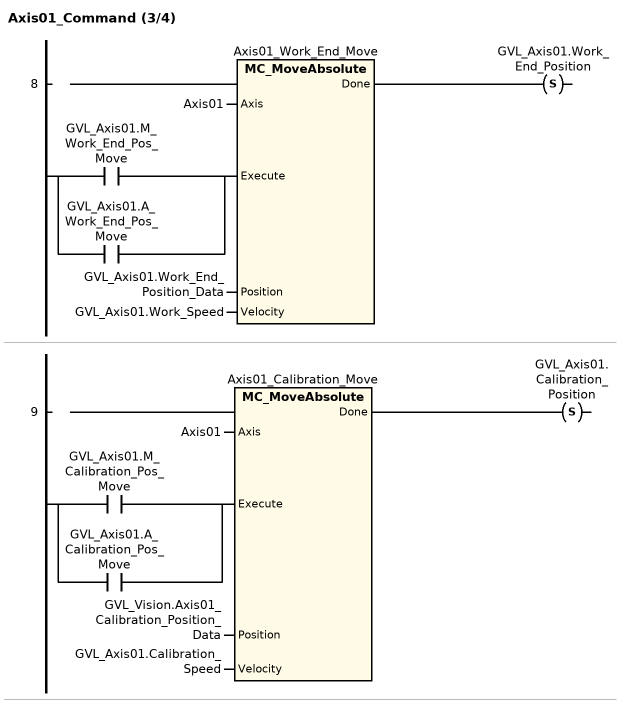
// NETWORK 8
Axis01_Work_End_Move(
    Axis := Axis01,
    Execute := GVL_Axis01.M_Work_End_Pos_Move OR GVL_Axis01.A_Work_End_Pos_Move,
    Position := GVL_Axis01.Work_End_Position_Data,
    Velocity := GVL_Axis01.Work_Speed); // MC_MoveAbsolute
GVL_Axis01.Work_End_Position S= Axis01_Work_End_Move.Done;

// NETWORK 9
Axis01_Calibration_Move(
    Axis := Axis01,
    Execute := GVL_Axis01.M_Calibration_Pos_Move OR GVL_Axis01.A_Calibration_Pos_Move,
    Position := GVL_Vision.Axis01_Calibration_Position_Data,
    Velocity := GVL_Axis01.Calibration_Speed); // MC_MoveAbsolute
GVL_Axis01.Calibration_Position S= Axis01_Calibration_Move.Done;

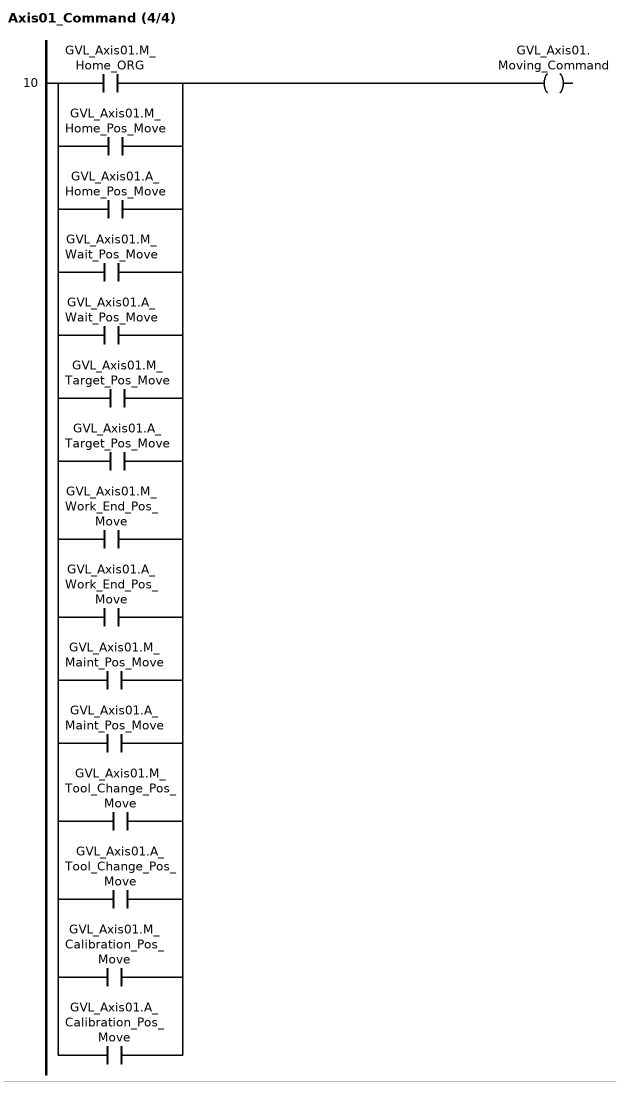
// NETWORK 10
GVL_Axis01.Moving_Command := GVL_Axis01.M_Home_ORG OR GVL_Axis01.M_Home_Pos_Move OR GVL_Axis01.A_Home_Pos_Move OR GVL_Axis01.M_Wait_Pos_Move OR GVL_Axis01.A_Wait_Pos_Move OR GVL_Axis01.M_Target_Pos_Move OR GVL_Axis01.A_Target_Pos_Move OR GVL_Axis01.M_Work_End_Pos_Move OR GVL_Axis01.A_Work_End_Pos_Move OR GVL_Axis01.M_Maint_Pos_Move OR GVL_Axis01.A_Maint_Pos_Move OR GVL_Axis01.M_Tool_Change_Pos_Move OR GVL_Axis01.A_Tool_Change_Pos_Move OR GVL_Axis01.M_Calibration_Pos_Move OR GVL_Axis01.A_Calibration_Pos_Move;

END_PROGRAM

// ---- POUs/FB_HomeBeforeMoveAX8000.TcPOU
FUNCTION_BLOCK FB_HomeBeforeMoveAX8000
VAR_IN_OUT
	AXIS : AXIS_REF;
END_VAR
VAR_INPUT
	Exectue : BOOL;	
	Homsensor : BOOL;
	LimitSensor : BOOL;
	HomePosition : LREAL;
	Channel : UINT :=1;

	// 0=FALSE, 1= TRUE
	InvertHomeSensorSearchDirection : WORD;
	// Velo
	HomeSensorVelocity : LREAL:=1;
	// 0=FALSE, 1= TRUE
	InvertSyncImpulseSearchDirection : WORD;
	// Velo
	SyncImpulseVelocity : LREAL:=1;
	
	// 0=FALSE, 1= TRUE
	InvertBeforeMoveDirection: WORD;
	// Velo
	BeforeMoveVelocity : LREAL:=1;
	
END_VAR
VAR_OUTPUT
	BUSY : BOOL;
	Error : BOOL;
	ErrorID : UDINT;
	ErrorStep : UDINT;
END_VAR
VAR
	//fbMC_WriteBoolParameter: MC_WriteBoolParameter;
	//fbMC_WriteParameter: MC_WriteParameter;
	//fbMC_MoveAbsolute: MC_MoveAbsolute;
	fbMC_MoveRelative: MC_MoveRelative;
	fbMC_Halt: MC_Halt;
	fbMC_Home : MC_Home;
	step: UDINT;
	fbADSWRITE_HomeSendsorBool: ADSWRITE;
	fbADSWRITE_HomeSendsorVeloLREAL: ADSWRITE;
	fbADSWRITE_SyncImpulseBool: ADSWRITE;
	fbADSWRITE_SyncImpulseVeloLREAL: ADSWRITE;
	fbR_TRIG: R_TRIG;
	
	NCPort: T_AmsPort := 501;
	fbTON: TON;
	WarningByte : BYTE:=2;
	ErrorByte : BYTE:=0;
	fbFB_CoEWrite_P_w: FB_CoEWrite;
	fbFB_CoEWrite_P_e: FB_CoEWrite;
	fbFB_CoEWrite_N_w: FB_CoEWrite;
	fbFB_CoEWrite_N_e: FB_CoEWrite;
END_VAR


CASE step OF
	0:
		fbR_TRIG(CLK:=Exectue);
		IF fbR_TRIG.Q THEN
			step:=10;
			fbMC_MoveRelative.Execute:=FALSE;
			fbMC_Home.Execute:=FALSE;
			fbMC_Halt.Execute:=FALSE;
			fbADSWRITE_HomeSendsorBool.WRITE:=FALSE;
			fbADSWRITE_HomeSendsorVeloLREAL.WRITE:=FALSE;
			fbADSWRITE_SyncImpulseBool.WRITE:=FALSE;
			fbADSWRITE_SyncImpulseVeloLREAL.WRITE:=FALSE;
			fbFB_CoEWrite_P_w.Execute:=FALSE;
			fbFB_CoEWrite_N_w.Execute:=FALSE;
			fbFB_CoEWrite_P_e.Execute:=FALSE;
			fbFB_CoEWrite_N_e.Execute:=FALSE;
			BUSY :=FALSE;
			Error :=FALSE;
			ErrorID :=0;
			ErrorStep :=0;
		END_IF
	10:
		fbFB_CoEWrite_P_w.Execute:=TRUE;
		fbFB_CoEWrite_N_w.Execute:=TRUE;
		step:=11;
	11:
		IF fbFB_CoEWrite_P_w.Busy=FALSE AND fbFB_CoEWrite_N_w.Busy=FALSE THEN
			IF fbFB_CoEWrite_P_w.Error THEN
				M_Error(_ErrorID:=fbFB_CoEWrite_P_w.AdsErrId,_ErrorStep:=step);
				step:=13;
			ELSIF fbFB_CoEWrite_N_w.Error THEN
				M_Error(_ErrorID:=fbFB_CoEWrite_N_w.AdsErrId,_ErrorStep:=step);
				step:=13;
			ELSE
				fbFB_CoEWrite_P_w.Execute:=FALSE;
				fbFB_CoEWrite_N_w.Execute:=FALSE;
				step:=15;
			END_IF
		END_IF
	
	//return start
	13:
		fbFB_CoEWrite_P_e.Execute:=TRUE;
		fbFB_CoEWrite_N_e.Execute:=TRUE;
		step:=14;
	14:
		IF fbFB_CoEWrite_P_e.Busy=FALSE AND fbFB_CoEWrite_N_e.Busy=FALSE THEN
			IF fbFB_CoEWrite_P_e.Error THEN
				M_Error(_ErrorID:=fbFB_CoEWrite_P_e.AdsErrId,_ErrorStep:=step);
			ELSIF fbFB_CoEWrite_N_e.Error THEN
				M_Error(_ErrorID:=fbFB_CoEWrite_N_e.AdsErrId,_ErrorStep:=step);
			ELSE
				fbFB_CoEWrite_P_e.Execute:=FALSE;
				fbFB_CoEWrite_N_e.Execute:=FALSE;
				step:=0;
			END_IF
		END_IF
	//return end

	15:
		IF InvertBeforeMoveDirection=1 THEN
			fbMC_MoveRelative.Distance := -1000000;
		ELSE
			fbMC_MoveRelative.Distance := 1000000;
		END_IF
		fbMC_MoveRelative.Velocity:=BeforeMoveVelocity;
		fbMC_MoveRelative.Execute:=TRUE;
		step:=20;
	20:
		IF fbMC_MoveRelative.Error=TRUE THEN;
			M_Error(_ErrorID:=fbMC_MoveRelative.ErrorID,_ErrorStep:=step);
			fbMC_MoveRelative.Execute:=FALSE;
			step:=13; // warning -> error
		ELSIF fbMC_MoveRelative.CommandAborted=TRUE THEN
			// jog 등 외부 명령이 이동을 가로챔 — 리밋 도달 불가. CoE 원복 후 재시작 가능하게 종료
			M_Error(_ErrorID:=16#FFFF0001,_ErrorStep:=step);
			fbMC_MoveRelative.Execute:=FALSE;
			step:=13; // warning -> error
		ELSE
			IF LimitSensor=TRUE OR ABS(AXIS.NcToPlc.PosDiff)>3 THEN
				//MC_SetAcceptBlockedDriveSignal(Axis := AXIS, Enable := FALSE);
				fbMC_Halt.Execute:=TRUE;
				step:=30;
			END_IF
		END_IF
		
	30:
		IF fbMC_Halt.Busy=FALSE THEN
			IF fbMC_Halt.Error=TRUE THEN
				M_Error(_ErrorID:=fbMC_Halt.ErrorID,_ErrorStep:=step);
				fbMC_Halt.Execute:=FALSE;
			ELSE
				fbMC_MoveRelative.Execute:=FALSE;
				fbMC_Halt.Execute:=FALSE;
				step:=200;
			END_IF
		END_IF
		
	200:
		fbADSWRITE_HomeSendsorBool.WRITE:=TRUE;
		M_NextStep10();
	210:
		IF fbADSWRITE_HomeSendsorBool.BUSY THEN
			IF fbADSWRITE_HomeSendsorBool.ERR=TRUE THEN
				M_Error(_ErrorID:=fbADSWRITE_HomeSendsorBool.ERRID,_ErrorStep:=step);
			ELSE
				fbADSWRITE_HomeSendsorBool.WRITE:=FALSE;
				M_NextStep10();
			END_IF
		END_IF
		
	220:
		fbADSWRITE_HomeSendsorVeloLREAL.WRITE:=TRUE;
		M_NextStep10();
	230:
		IF fbADSWRITE_HomeSendsorVeloLREAL.BUSY THEN
			IF fbADSWRITE_HomeSendsorVeloLREAL.ERR=TRUE THEN
				M_Error(_ErrorID:=fbADSWRITE_HomeSendsorVeloLREAL.ERRID,_ErrorStep:=step);
			ELSE
				fbADSWRITE_HomeSendsorVeloLREAL.WRITE:=FALSE;
				M_NextStep10();
			END_IF
		END_IF
	
	240:
		fbADSWRITE_SyncImpulseBool.WRITE:=TRUE;
		M_NextStep10();
	250:
		IF fbADSWRITE_SyncImpulseBool.BUSY THEN
			IF fbADSWRITE_SyncImpulseBool.ERR=TRUE THEN
				M_Error(_ErrorID:=fbADSWRITE_SyncImpulseBool.ERRID,_ErrorStep:=step);
			ELSE
				fbADSWRITE_SyncImpulseBool.WRITE:=FALSE;
				M_NextStep10();
			END_IF
		END_IF
	
	260:
		fbADSWRITE_SyncImpulseVeloLREAL.WRITE:=TRUE;
		M_NextStep10();
	270:
		IF fbADSWRITE_SyncImpulseVeloLREAL.BUSY THEN
			IF fbADSWRITE_SyncImpulseVeloLREAL.ERR=TRUE THEN
				M_Error(_ErrorID:=fbADSWRITE_SyncImpulseVeloLREAL.ERRID,_ErrorStep:=step);
			ELSE
				fbADSWRITE_SyncImpulseVeloLREAL.WRITE:=FALSE;
				M_NextStep10();
			END_IF
		END_IF
	280:
		fbTON(IN:=TRUE,PT:=T#0.5S);
		IF fbTON.q THEN
			fbTON(IN:=FALSE);
			IF fbADSWRITE_HomeSendsorBool.ERR=TRUE THEN
				M_Error(_ErrorID:=fbADSWRITE_HomeSendsorBool.ERRID,_ErrorStep:=210);
			ELSIF fbADSWRITE_HomeSendsorVeloLREAL.ERR=TRUE THEN;
				M_Error(_ErrorID:=fbADSWRITE_HomeSendsorVeloLREAL.ERRID,_ErrorStep:=230);
			ELSIF fbADSWRITE_SyncImpulseBool.ERR=TRUE THEN;
				M_Error(_ErrorID:=fbADSWRITE_SyncImpulseBool.ERRID,_ErrorStep:=250);
			ELSIF fbADSWRITE_SyncImpulseVeloLREAL.ERR=TRUE THEN;
				M_Error(_ErrorID:=fbADSWRITE_SyncImpulseVeloLREAL.ERRID,_ErrorStep:=270);
			ELSE
				step:=300;
			END_IF
		END_IF
	
	300:
		fbMC_Home.Execute:=TRUE;
		M_NextStep10();
	310:
		IF fbMC_Home.Busy=FALSE THEN
			fbTON(IN:=TRUE,PT:=T#0.5S);
			IF fbTON.q THEN
				fbTON(IN:=FALSE);
				IF fbMC_Home.Error=TRUE THEN
					M_Error(_ErrorID:=fbMC_Home.ErrorID,_ErrorStep:=step);
					step:=13; // CoE 리밋 반응 원복 후 종료
				ELSIF fbMC_Home.CommandAborted=TRUE THEN
					// jog 등이 홈을 가로챔 — 성공으로 오인 금지, 미완료 에러 처리
					M_Error(_ErrorID:=16#FFFF0002,_ErrorStep:=step);
					step:=13; // CoE 리밋 반응 원복 후 종료
				ELSE
					step:=320;
				END_IF
				fbMC_Home.Execute:=FALSE;
			END_IF
		END_IF
	320:
		fbFB_CoEWrite_P_e.Execute:=TRUE;
		fbFB_CoEWrite_N_e.Execute:=TRUE;
		step:=330;
	330:
		IF fbFB_CoEWrite_P_e.Busy=FALSE AND fbFB_CoEWrite_N_e.Busy=FALSE THEN
			IF fbFB_CoEWrite_P_e.Error THEN
				M_Error(_ErrorID:=fbFB_CoEWrite_P_e.AdsErrId,_ErrorStep:=step);
			ELSIF fbFB_CoEWrite_N_e.Error THEN
				M_Error(_ErrorID:=fbFB_CoEWrite_N_e.AdsErrId,_ErrorStep:=step);
			ELSE
				fbFB_CoEWrite_P_e.Execute:=FALSE;
				fbFB_CoEWrite_N_e.Execute:=FALSE;
				step:=0;
			END_IF
		END_IF
END_CASE
BUSY := Step<>0;

	
fbADSWRITE_HomeSendsorBool(
	PORT:= NCPort, 
	IDXGRP:= 16#5000+AXIS.NcToPlc.AxisId, 
	IDXOFFS:= 16#101, 
	LEN:= SIZEOF(InvertHomeSensorSearchDirection), 
	SRCADDR:= ADR(InvertHomeSensorSearchDirection));
fbADSWRITE_HomeSendsorVeloLREAL(
	PORT:= NCPort, 
	IDXGRP:= 16#4000+AXIS.NcToPlc.AxisId, 
	IDXOFFS:= 16#6, 
	LEN:= SIZEOF(HomeSensorVelocity), 
	SRCADDR:= ADR(HomeSensorVelocity));
fbADSWRITE_SyncImpulseBool(
	PORT:= NCPort, 
	IDXGRP:= 16#5000+AXIS.NcToPlc.AxisId, 
	IDXOFFS:= 16#102, 
	LEN:= SIZEOF(InvertSyncImpulseSearchDirection), 
	SRCADDR:= ADR(InvertSyncImpulseSearchDirection));
fbADSWRITE_SyncImpulseVeloLREAL(
	PORT:= NCPort, 
	IDXGRP:= 16#4000+AXIS.NcToPlc.AxisId, 
	IDXOFFS:= 16#7, 
	LEN:= SIZEOF(SyncImpulseVelocity), 
	SRCADDR:= ADR(SyncImpulseVelocity));
	
fbMC_MoveRelative(
	Axis:= AXIS, 
	Execute:= , 
	Distance:= , 
	Velocity:= , 
	Acceleration:= , 
	Deceleration:= , 
	Jerk:= , 
	BufferMode:= , 
	Options:= , 
	Done=> , 
	Busy=> , 
	Active=> , 
	CommandAborted=> , 
	Error=> , 
	ErrorID=> );
fbMC_Halt(
	Axis:= AXIS, 
	Execute:= , 
	Deceleration:= , 
	Jerk:= , 
	BufferMode:= , 
	Options:= , 
	Done=> , 
	Busy=> , 
	Active=> , 
	CommandAborted=> , 
	Error=> , 
	ErrorID=> );
fbMC_Home(
	Axis:= AXIS, 
	Execute:= , 
	Position:= HomePosition, 
	HomingMode:= , 
	BufferMode:= , 
	Options:= , 
	bCalibrationCam:= Homsensor, 
	Done=> , 
	Busy=> , 
	Active=> , 
	CommandAborted=> , 
	Error=> , 
	ErrorID=> );
IF Channel=1 THEN
	fbFB_CoEWrite_P_w(
		Axis:= AXIS, 
		NetId:= , 
		Index:= 16#3002, 
		SubIndex:= 16#03, 
		pSrcBuf:= ADR(WarningByte), 
		BufLen:= SIZEOF(WarningByte));
	fbFB_CoEWrite_P_e(
		Axis:= AXIS, 
		NetId:= , 
		Index:= 16#3002, 
		SubIndex:= 16#03, 
		pSrcBuf:= ADR(ErrorByte), 
		BufLen:= SIZEOF(ErrorByte));
	
	fbFB_CoEWrite_N_w(
		Axis:= AXIS, 
		NetId:= , 
		Index:= 16#3003, 
		SubIndex:= 16#03, 
		pSrcBuf:= ADR(WarningByte), 
		BufLen:= SIZEOF(WarningByte));
	fbFB_CoEWrite_N_e(
		Axis:= AXIS, 
		NetId:= , 
		Index:= 16#3003, 
		SubIndex:= 16#03, 
		pSrcBuf:= ADR(ErrorByte), 
		BufLen:= SIZEOF(ErrorByte));
ELSIF Channel=2 THEN
	fbFB_CoEWrite_P_w(
		Axis:= AXIS, 
		NetId:= , 
		Index:= 16#3402, 
		SubIndex:= 16#03, 
		pSrcBuf:= ADR(WarningByte), 
		BufLen:= SIZEOF(WarningByte));
	fbFB_CoEWrite_P_e(
		Axis:= AXIS, 
		NetId:= , 
		Index:= 16#3402, 
		SubIndex:= 16#03, 
		pSrcBuf:= ADR(ErrorByte), 
		BufLen:= SIZEOF(ErrorByte));
	
	fbFB_CoEWrite_N_w(
		Axis:= AXIS, 
		NetId:= , 
		Index:= 16#3403, 
		SubIndex:= 16#03, 
		pSrcBuf:= ADR(WarningByte), 
		BufLen:= SIZEOF(WarningByte));
	fbFB_CoEWrite_N_e(
		Axis:= AXIS, 
		NetId:= , 
		Index:= 16#3403, 
		SubIndex:= 16#03, 
		pSrcBuf:= ADR(ErrorByte), 
		BufLen:= SIZEOF(ErrorByte));
END_IF

METHOD M_Error : BOOL
VAR_INPUT
	_ErrorID : UDINT;
	_ErrorStep: UDINT;
END_VAR
step:=0;
Error :=TRUE;
ErrorID := _ErrorID;
ErrorStep := _ErrorStep;
END_METHOD

METHOD M_NextStep10 : BOOL
VAR_INPUT
END_VAR
step:=step+10;
END_METHOD

END_FUNCTION_BLOCK

// ---- POUs/Axis01_R/Axis01_Manual.TcPOU
PROGRAM Axis01_Manual
VAR
//System_Bit
	Always_ON	:	BOOL	:=TRUE	;//상시 ON 
	Always_OFF	:	BOOL	:=FALSE	;//상시 OFF
END_VAR
VAR // added by the converter: edge detectors and wires of the graphical bodies
    _rt1, _rt2, _rt3 : R_TRIG;
END_VAR

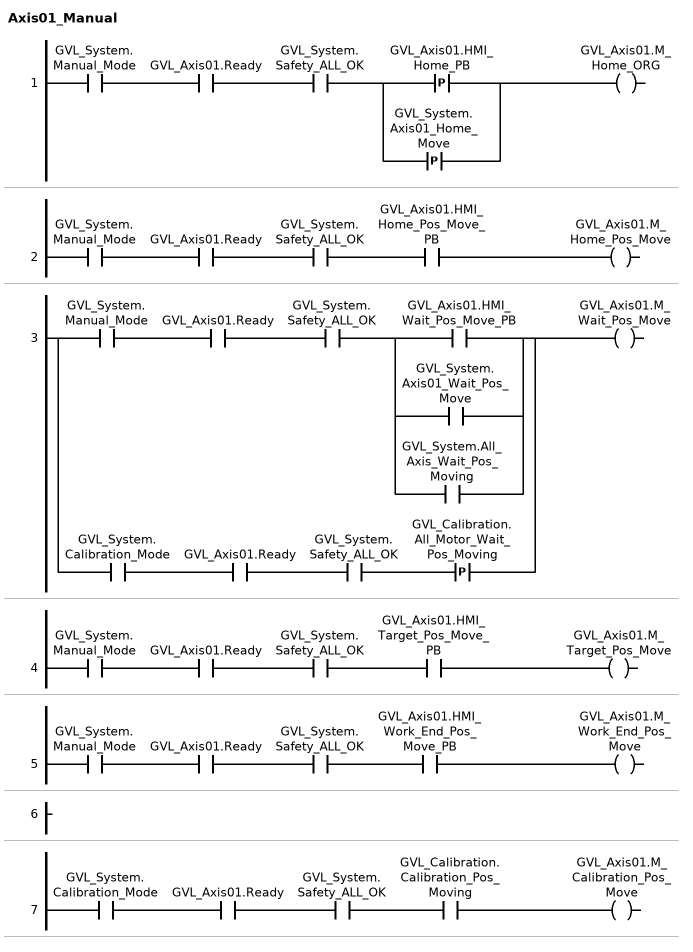
// NETWORK 1
_rt1(CLK := GVL_Axis01.HMI_Home_PB);
_rt2(CLK := GVL_System.Axis01_Home_Move);
GVL_Axis01.M_Home_ORG := GVL_System.Manual_Mode AND GVL_Axis01.Ready AND GVL_System.Safety_ALL_OK AND (_rt1.Q OR _rt2.Q);

// NETWORK 2
GVL_Axis01.M_Home_Pos_Move := GVL_System.Manual_Mode AND GVL_Axis01.Ready AND GVL_System.Safety_ALL_OK AND GVL_Axis01.HMI_Home_Pos_Move_PB;

// NETWORK 3
_rt3(CLK := GVL_Calibration.All_Motor_Wait_Pos_Moving);
GVL_Axis01.M_Wait_Pos_Move := GVL_System.Manual_Mode AND GVL_Axis01.Ready AND GVL_System.Safety_ALL_OK AND (GVL_Axis01.HMI_Wait_Pos_Move_PB OR GVL_System.Axis01_Wait_Pos_Move OR GVL_System.All_Axis_Wait_Pos_Moving) OR GVL_System.Calibration_Mode AND GVL_Axis01.Ready AND GVL_System.Safety_ALL_OK AND _rt3.Q;

// NETWORK 4
GVL_Axis01.M_Target_Pos_Move := GVL_System.Manual_Mode AND GVL_Axis01.Ready AND GVL_System.Safety_ALL_OK AND GVL_Axis01.HMI_Target_Pos_Move_PB;

// NETWORK 5
GVL_Axis01.M_Work_End_Pos_Move := GVL_System.Manual_Mode AND GVL_Axis01.Ready AND GVL_System.Safety_ALL_OK AND GVL_Axis01.HMI_Work_End_Pos_Move_PB;

// NETWORK 6

// NETWORK 7
GVL_Axis01.M_Calibration_Pos_Move := GVL_System.Calibration_Mode AND GVL_Axis01.Ready AND GVL_System.Safety_ALL_OK AND GVL_Calibration.Calibration_Pos_Moving;

END_PROGRAM

// ---- POUs/Axis01_R/Axis01_Auto.TcPOU
PROGRAM Axis01_Auto
VAR
//System_Bit
	Always_ON	:	BOOL	:=TRUE	;//상시 ON 
	Always_OFF	:	BOOL	:=FALSE	;//상시 OFF
END_VAR

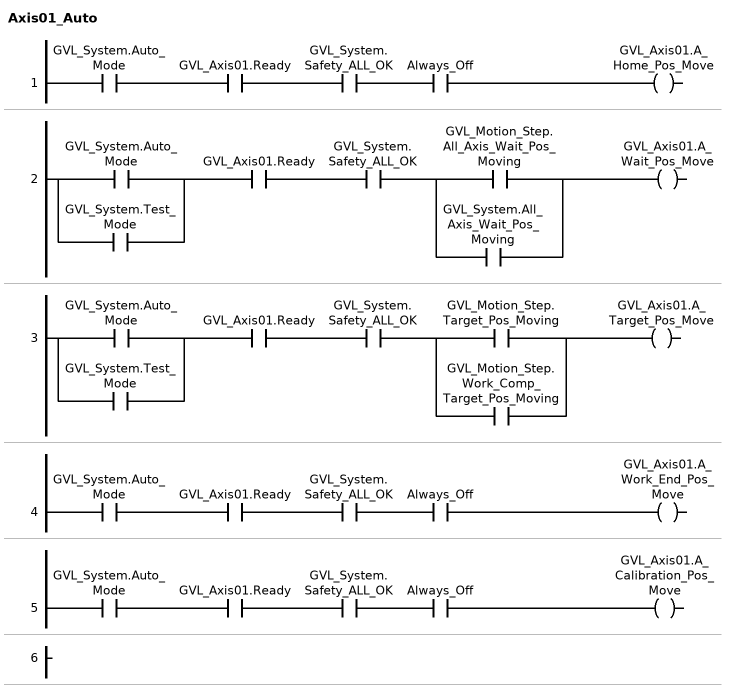
// NETWORK 1
GVL_Axis01.A_Home_Pos_Move := GVL_System.Auto_Mode AND GVL_Axis01.Ready AND GVL_System.Safety_ALL_OK AND Always_Off;

// NETWORK 2
GVL_Axis01.A_Wait_Pos_Move := (GVL_System.Auto_Mode OR GVL_System.Test_Mode) AND GVL_Axis01.Ready AND GVL_System.Safety_ALL_OK AND (GVL_Motion_Step.All_Axis_Wait_Pos_Moving OR GVL_System.All_Axis_Wait_Pos_Moving);

// NETWORK 3
GVL_Axis01.A_Target_Pos_Move := (GVL_System.Auto_Mode OR GVL_System.Test_Mode) AND GVL_Axis01.Ready AND GVL_System.Safety_ALL_OK AND (GVL_Motion_Step.Target_Pos_Moving OR GVL_Motion_Step.Work_Comp_Target_Pos_Moving);

// NETWORK 4
GVL_Axis01.A_Work_End_Pos_Move := GVL_System.Auto_Mode AND GVL_Axis01.Ready AND GVL_System.Safety_ALL_OK AND Always_Off;

// NETWORK 5
GVL_Axis01.A_Calibration_Pos_Move := GVL_System.Auto_Mode AND GVL_Axis01.Ready AND GVL_System.Safety_ALL_OK AND Always_Off;

// NETWORK 6

END_PROGRAM

// ---- POUs/Axis01_R/Axis01_Alarm.TcPOU
PROGRAM Axis01_Alarm
VAR
//System_Bit
	Always_ON	:	BOOL	:=TRUE	;//상시 ON 
	Always_OFF	:	BOOL	:=FALSE	;//상시 OFF
END_VAR

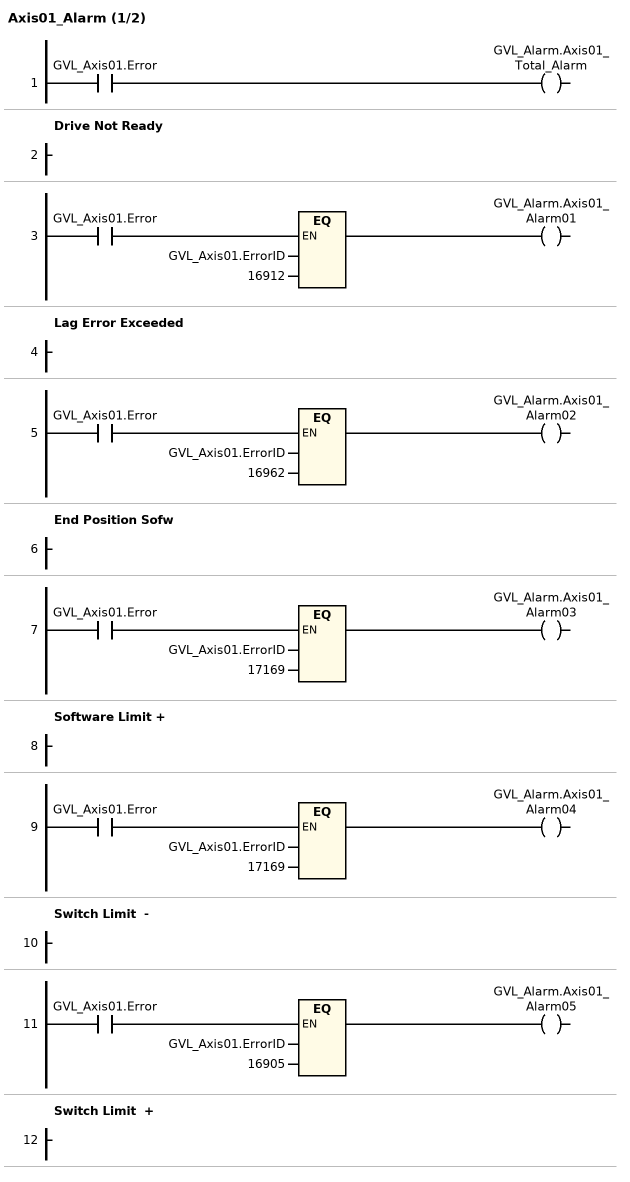
// NETWORK 1
GVL_Alarm.Axis01_Total_Alarm := GVL_Axis01.Error;

// NETWORK 2: Drive Not Ready

// NETWORK 3
GVL_Alarm.Axis01_Alarm01 := GVL_Axis01.Error AND GVL_Axis01.ErrorID = 16912;

// NETWORK 4: Lag Error Exceeded

// NETWORK 5
GVL_Alarm.Axis01_Alarm02 := GVL_Axis01.Error AND GVL_Axis01.ErrorID = 16962;

// NETWORK 6: End Position Sofw

// NETWORK 7
GVL_Alarm.Axis01_Alarm03 := GVL_Axis01.Error AND GVL_Axis01.ErrorID = 17169;

// NETWORK 8: Software Limit +

// NETWORK 9
GVL_Alarm.Axis01_Alarm04 := GVL_Axis01.Error AND GVL_Axis01.ErrorID = 17169;

// NETWORK 10: Switch Limit -

// NETWORK 11
GVL_Alarm.Axis01_Alarm05 := GVL_Axis01.Error AND GVL_Axis01.ErrorID = 16905;

// NETWORK 12: Switch Limit +

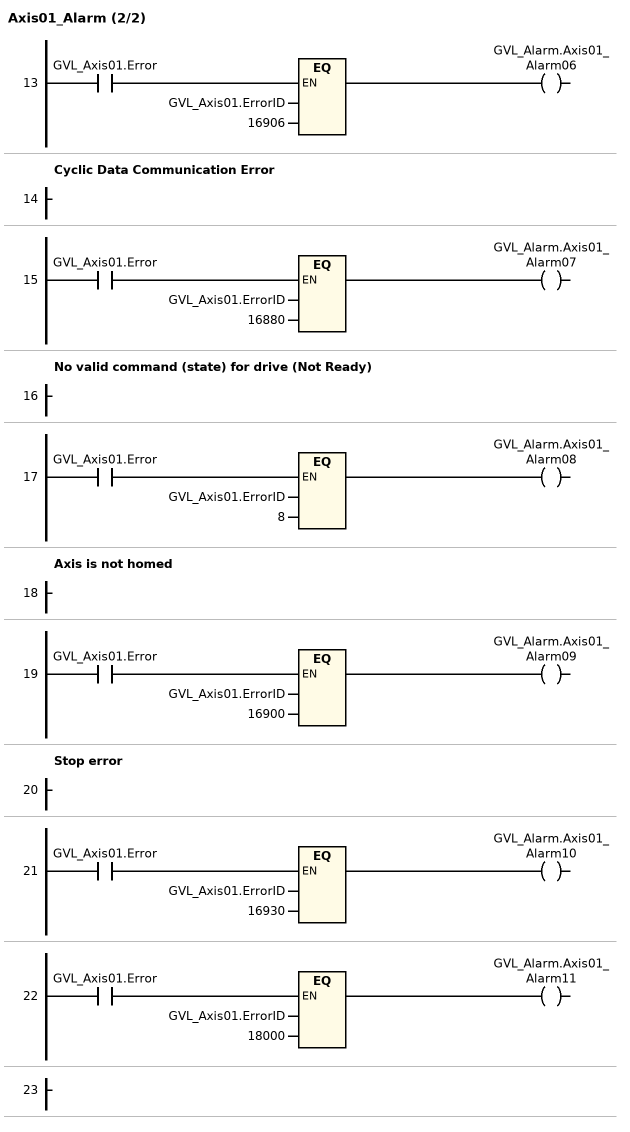
// NETWORK 13
GVL_Alarm.Axis01_Alarm06 := GVL_Axis01.Error AND GVL_Axis01.ErrorID = 16906;

// NETWORK 14: Cyclic Data Communication Error

// NETWORK 15
GVL_Alarm.Axis01_Alarm07 := GVL_Axis01.Error AND GVL_Axis01.ErrorID = 16880;

// NETWORK 16: No valid command (state) for drive (Not Ready)

// NETWORK 17
GVL_Alarm.Axis01_Alarm08 := GVL_Axis01.Error AND GVL_Axis01.ErrorID = 8;

// NETWORK 18: Axis is not homed

// NETWORK 19
GVL_Alarm.Axis01_Alarm09 := GVL_Axis01.Error AND GVL_Axis01.ErrorID = 16900;

// NETWORK 20: Stop error

// NETWORK 21
GVL_Alarm.Axis01_Alarm10 := GVL_Axis01.Error AND GVL_Axis01.ErrorID = 16930;

// NETWORK 22
GVL_Alarm.Axis01_Alarm11 := GVL_Axis01.Error AND GVL_Axis01.ErrorID = 18000;

// NETWORK 23

END_PROGRAM

// ---- POUs/Axis02_X/Axis02_Status.TcPOU
PROGRAM Axis02_Status
VAR
//System_Bit
	Always_ON	:	BOOL	:=TRUE	;//상시 ON 
	Always_OFF	:	BOOL	:=FALSE	;//상시 OFF
	
//Motor_Command
	Axis02_Status_01: MC_ReadStatus;
	Axis02_Position_Read_01: MC_ReadActualPosition;
	Axis02_Velocity_Read_01: MC_ReadActualVelocity;
	Axis02_Reset_01: MC_Reset;
	Axis02_Stop_01: MC_Stop;
END_VAR

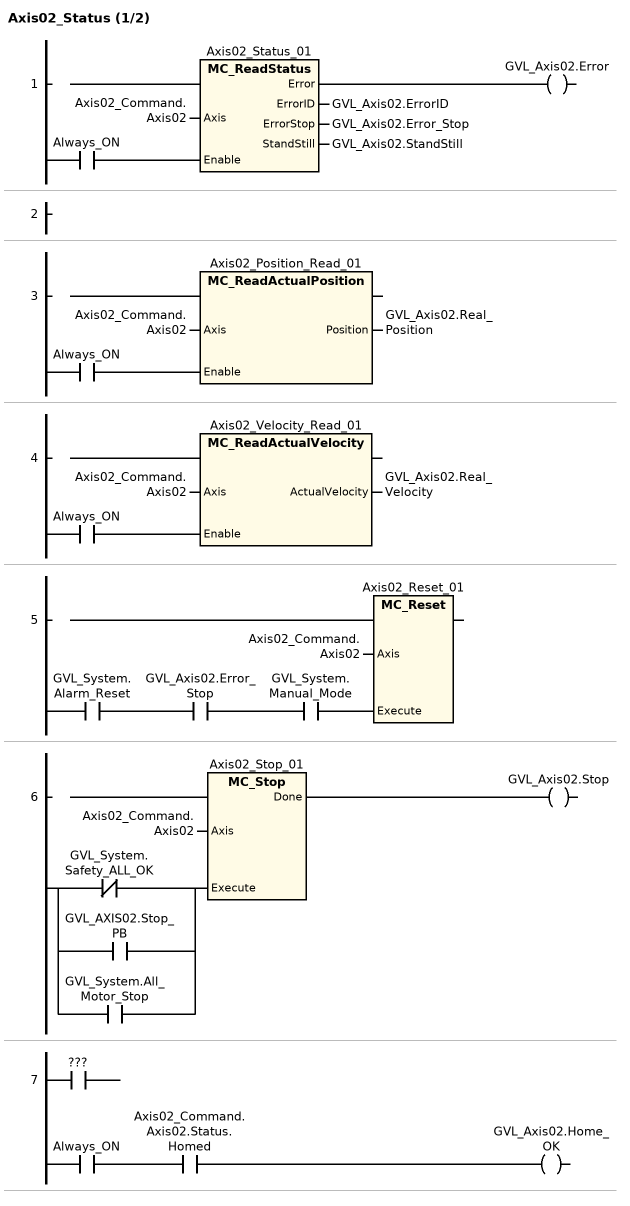
// NETWORK 1
Axis02_Status_01(
    Axis := Axis02_Command.Axis02,
    Enable := Always_ON,
    Error => GVL_Axis02.Error,
    ErrorID => GVL_Axis02.ErrorID,
    ErrorStop => GVL_Axis02.Error_Stop,
    StandStill => GVL_Axis02.StandStill); // MC_ReadStatus

// NETWORK 2

// NETWORK 3
Axis02_Position_Read_01(
    Axis := Axis02_Command.Axis02,
    Enable := Always_ON,
    Position => GVL_Axis02.Real_Position); // MC_ReadActualPosition

// NETWORK 4
Axis02_Velocity_Read_01(
    Axis := Axis02_Command.Axis02,
    Enable := Always_ON,
    ActualVelocity => GVL_Axis02.Real_Velocity); // MC_ReadActualVelocity

// NETWORK 5
Axis02_Reset_01(Axis := Axis02_Command.Axis02, Execute := GVL_System.Alarm_Reset AND GVL_Axis02.Error_Stop AND GVL_System.Manual_Mode); // MC_Reset

// NETWORK 6
Axis02_Stop_01(Axis := Axis02_Command.Axis02, Execute := NOT GVL_System.Safety_ALL_OK OR GVL_AXIS02.Stop_PB OR GVL_System.All_Motor_Stop); // MC_Stop
GVL_Axis02.Stop := Axis02_Stop_01.Done;

// NETWORK 7
GVL_Axis02.Home_OK := Always_ON AND Axis02_Command.Axis02.Status.Homed;

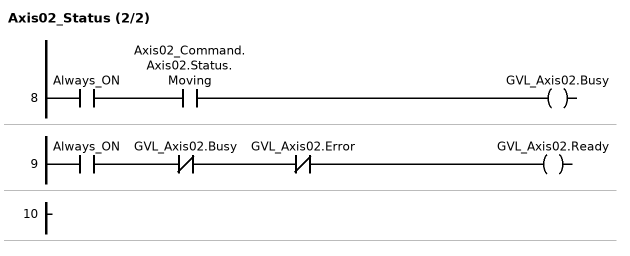
// NETWORK 8
GVL_Axis02.Busy := Always_ON AND Axis02_Command.Axis02.Status.Moving;

// NETWORK 9
GVL_Axis02.Ready := Always_ON AND NOT GVL_Axis02.Busy AND NOT GVL_Axis02.Error;

// NETWORK 10

END_PROGRAM

// ---- POUs/Axis02_X/Axis02_Command.TcPOU
PROGRAM Axis02_Command
VAR
//System_Bit
	Always_ON	:	BOOL	:=TRUE	;//상시 ON 
	Always_OFF	:	BOOL	:=FALSE	;//상시 OFF

//Motor_Command
	Axis02: AXIS_REF;											//회전축
	Axis02_MC_Power: MC_Power;
	Axis02_MC_Home: FB_HomeBeforeMoveAX8000:=(channel:=2);
	Axis02_Jog: MC_Jog;
	Axis02_Home_Pos_Move: MC_MoveAbsolute;
	Axis02_Wait_Pos_Move: MC_MoveAbsolute;
	Axis02_Target_Pos_Move: MC_MoveAbsolute;
	Axi02_Work_End_Move: MC_GearInVelo;
	Work_Offset_Move: MC_MoveSuperImposed;
	Axis02_Work_End_Comp: MC_GearOut;
	Axis02_Maint_Move: MC_MoveAbsolute;
	Axis02_Tool_Change: MC_MoveAbsolute;
	Axis02_Calibration: MC_MoveAbsolute;	



	
	Test002: BOOL;
	Test001: BOOL;

	Axis02_Stop_02: MC_Stop;
	Work_Comp: BOOL;
	Work_Stop: BOOL;


	Timer01: TON;
	Axis02_Work_End_Move_Test: MC_MoveAbsolute;
	Encoder_Real_Velocity: LREAL;
	MC_GearInPos_0: MC_GearInPos;
	keb_X: BOOL;
	Axis02_ku_Pos_Move: MC_MoveAbsolute;
	keb_X_data_PB: BOOL;
END_VAR
VAR // added by the converter: edge detectors and wires of the graphical bodies
    _rt1, _rt2 : R_TRIG;
END_VAR

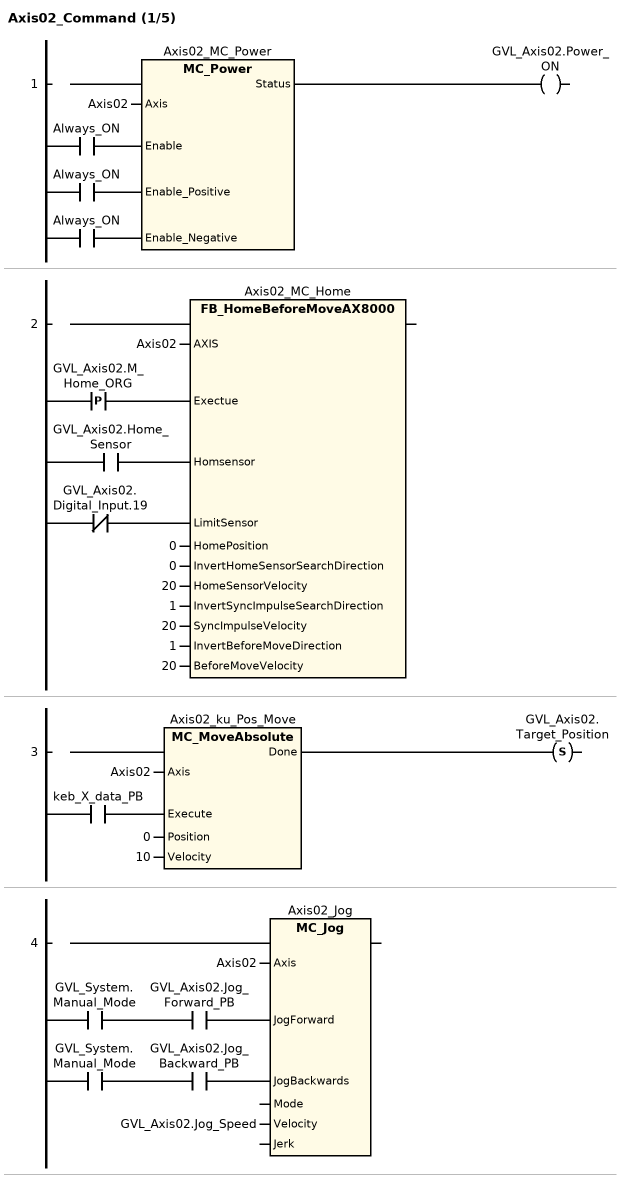
// NETWORK 1
Axis02_MC_Power(
    Axis := Axis02,
    Enable := Always_ON,
    Enable_Positive := Always_ON,
    Enable_Negative := Always_ON); // MC_Power
GVL_Axis02.Power_ON := Axis02_MC_Power.Status;

// NETWORK 2
_rt1(CLK := GVL_Axis02.M_Home_ORG);
Axis02_MC_Home(
    AXIS := Axis02,
    Exectue := _rt1.Q,
    Homsensor := GVL_Axis02.Home_Sensor,
    LimitSensor := NOT GVL_Axis02.Digital_Input.19,
    HomePosition := 0,
    InvertHomeSensorSearchDirection := 0,
    HomeSensorVelocity := 20,
    InvertSyncImpulseSearchDirection := 1,
    SyncImpulseVelocity := 20,
    InvertBeforeMoveDirection := 1,
    BeforeMoveVelocity := 20); // FB_HomeBeforeMoveAX8000

// NETWORK 3
Axis02_ku_Pos_Move(Axis := Axis02, Execute := keb_X_data_PB, Position := 0, Velocity := 10); // MC_MoveAbsolute
GVL_Axis02.Target_Position S= Axis02_ku_Pos_Move.Done;

// NETWORK 4
Axis02_Jog(
    Axis := Axis02,
    JogForward := GVL_System.Manual_Mode AND GVL_Axis02.Jog_Forward_PB,
    JogBackwards := GVL_System.Manual_Mode AND GVL_Axis02.Jog_Backward_PB,
    Velocity := GVL_Axis02.Jog_Speed); // MC_Jog

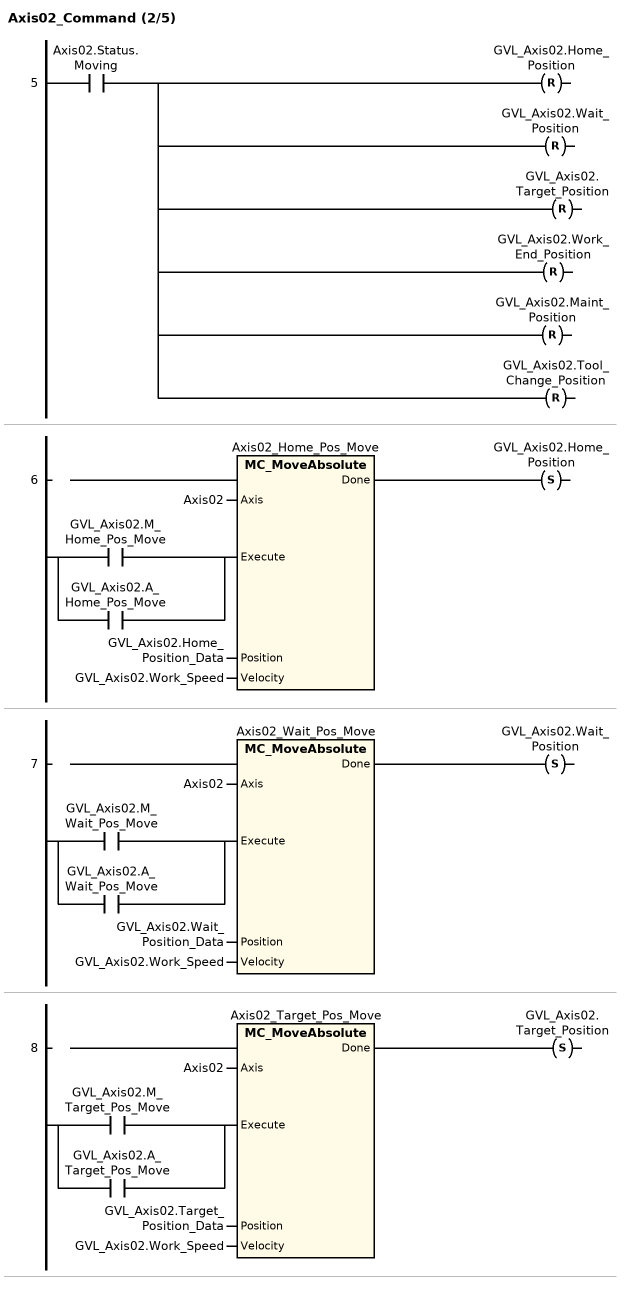
// NETWORK 5
GVL_Axis02.Home_Position R= Axis02.Status.Moving;
GVL_Axis02.Wait_Position R= Axis02.Status.Moving;
GVL_Axis02.Target_Position R= Axis02.Status.Moving;
GVL_Axis02.Work_End_Position R= Axis02.Status.Moving;
GVL_Axis02.Maint_Position R= Axis02.Status.Moving;
GVL_Axis02.Tool_Change_Position R= Axis02.Status.Moving;

// NETWORK 6
Axis02_Home_Pos_Move(
    Axis := Axis02,
    Execute := GVL_Axis02.M_Home_Pos_Move OR GVL_Axis02.A_Home_Pos_Move,
    Position := GVL_Axis02.Home_Position_Data,
    Velocity := GVL_Axis02.Work_Speed); // MC_MoveAbsolute
GVL_Axis02.Home_Position S= Axis02_Home_Pos_Move.Done;

// NETWORK 7
Axis02_Wait_Pos_Move(
    Axis := Axis02,
    Execute := GVL_Axis02.M_Wait_Pos_Move OR GVL_Axis02.A_Wait_Pos_Move,
    Position := GVL_Axis02.Wait_Position_Data,
    Velocity := GVL_Axis02.Work_Speed); // MC_MoveAbsolute
GVL_Axis02.Wait_Position S= Axis02_Wait_Pos_Move.Done;

// NETWORK 8
Axis02_Target_Pos_Move(
    Axis := Axis02,
    Execute := GVL_Axis02.M_Target_Pos_Move OR GVL_Axis02.A_Target_Pos_Move,
    Position := GVL_Axis02.Target_Position_Data,
    Velocity := GVL_Axis02.Work_Speed); // MC_MoveAbsolute
GVL_Axis02.Target_Position S= Axis02_Target_Pos_Move.Done;

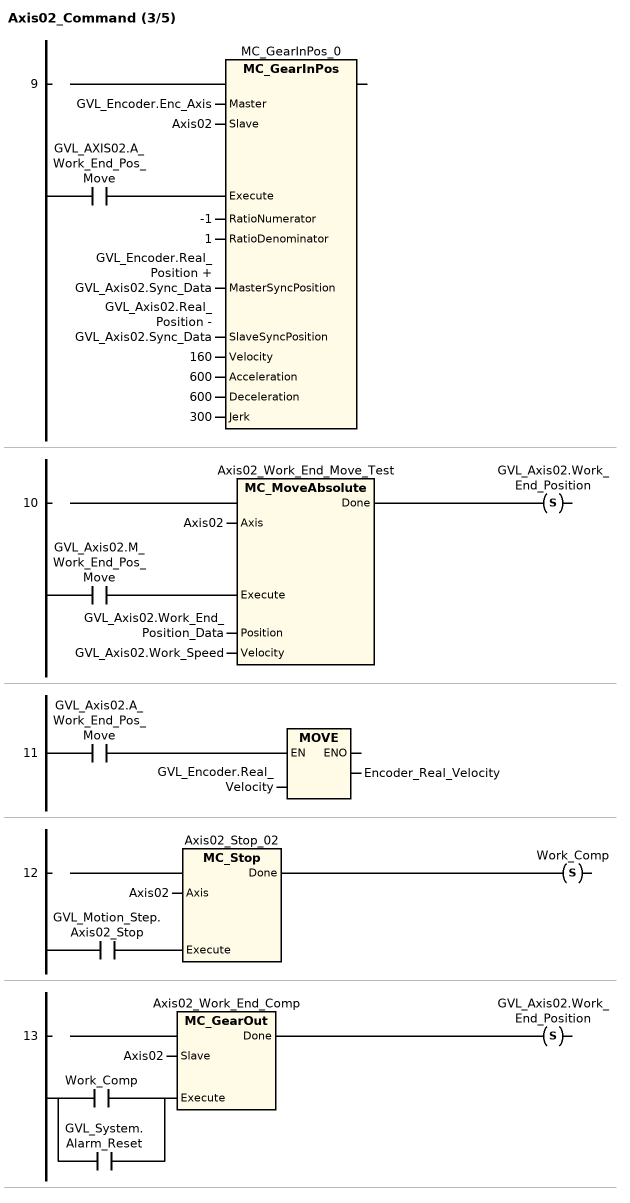
// NETWORK 9
MC_GearInPos_0(
    Master := GVL_Encoder.Enc_Axis,
    Slave := Axis02,
    Execute := GVL_AXIS02.A_Work_End_Pos_Move,
    RatioNumerator := -1,
    RatioDenominator := 1,
    MasterSyncPosition := GVL_Encoder.Real_Position + GVL_Axis02.Sync_Data,
    SlaveSyncPosition := GVL_Axis02.Real_Position - GVL_Axis02.Sync_Data,
    Velocity := 160,
    Acceleration := 600,
    Deceleration := 600,
    Jerk := 300); // MC_GearInPos

// NETWORK 10
Axis02_Work_End_Move_Test(
    Axis := Axis02,
    Execute := GVL_Axis02.M_Work_End_Pos_Move,
    Position := GVL_Axis02.Work_End_Position_Data,
    Velocity := GVL_Axis02.Work_Speed); // MC_MoveAbsolute
GVL_Axis02.Work_End_Position S= Axis02_Work_End_Move_Test.Done;

// NETWORK 11
IF GVL_Axis02.A_Work_End_Pos_Move THEN Encoder_Real_Velocity := GVL_Encoder.Real_Velocity; END_IF

// NETWORK 12
Axis02_Stop_02(Axis := Axis02, Execute := GVL_Motion_Step.Axis02_Stop); // MC_Stop
Work_Comp S= Axis02_Stop_02.Done;

// NETWORK 13
Axis02_Work_End_Comp(Slave := Axis02, Execute := Work_Comp OR GVL_System.Alarm_Reset); // MC_GearOut
GVL_Axis02.Work_End_Position S= Axis02_Work_End_Comp.Done;

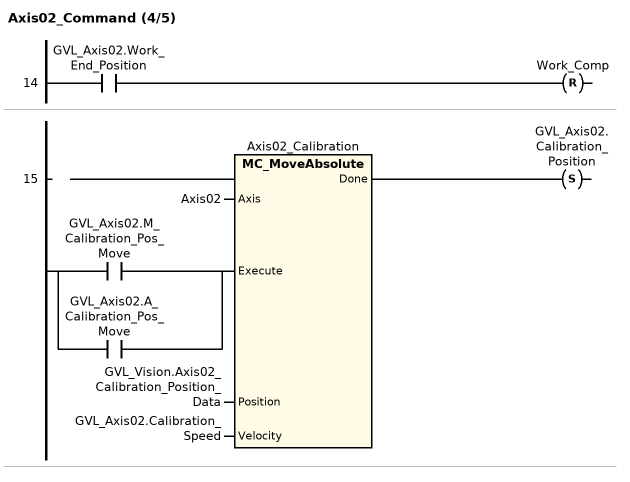
// NETWORK 14
Work_Comp R= GVL_Axis02.Work_End_Position;

// NETWORK 15
Axis02_Calibration(
    Axis := Axis02,
    Execute := GVL_Axis02.M_Calibration_Pos_Move OR GVL_Axis02.A_Calibration_Pos_Move,
    Position := GVL_Vision.Axis02_Calibration_Position_Data,
    Velocity := GVL_Axis02.Calibration_Speed); // MC_MoveAbsolute
GVL_Axis02.Calibration_Position S= Axis02_Calibration.Done;

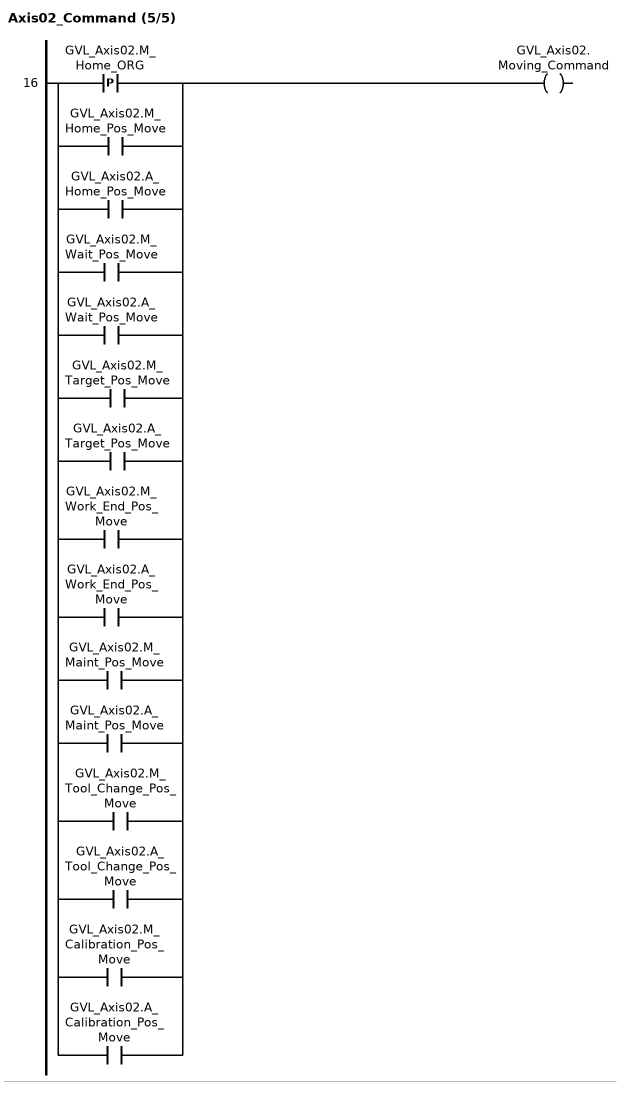
// NETWORK 16
_rt2(CLK := GVL_Axis02.M_Home_ORG);
GVL_Axis02.Moving_Command := _rt2.Q OR GVL_Axis02.M_Home_Pos_Move OR GVL_Axis02.A_Home_Pos_Move OR GVL_Axis02.M_Wait_Pos_Move OR GVL_Axis02.A_Wait_Pos_Move OR GVL_Axis02.M_Target_Pos_Move OR GVL_Axis02.A_Target_Pos_Move OR GVL_Axis02.M_Work_End_Pos_Move OR GVL_Axis02.A_Work_End_Pos_Move OR GVL_Axis02.M_Maint_Pos_Move OR GVL_Axis02.A_Maint_Pos_Move OR GVL_Axis02.M_Tool_Change_Pos_Move OR GVL_Axis02.A_Tool_Change_Pos_Move OR GVL_Axis02.M_Calibration_Pos_Move OR GVL_Axis02.A_Calibration_Pos_Move;

END_PROGRAM

// ---- POUs/Axis02_X/Axis02_Manual.TcPOU
PROGRAM Axis02_Manual
VAR
//System_Bit
	Always_ON	:	BOOL	:=TRUE	;//상시 ON 
	Always_OFF	:	BOOL	:=FALSE	;//상시 OFF
END_VAR
VAR // added by the converter: edge detectors and wires of the graphical bodies
    _rt1, _rt2, _rt3, _rt4 : R_TRIG;
END_VAR

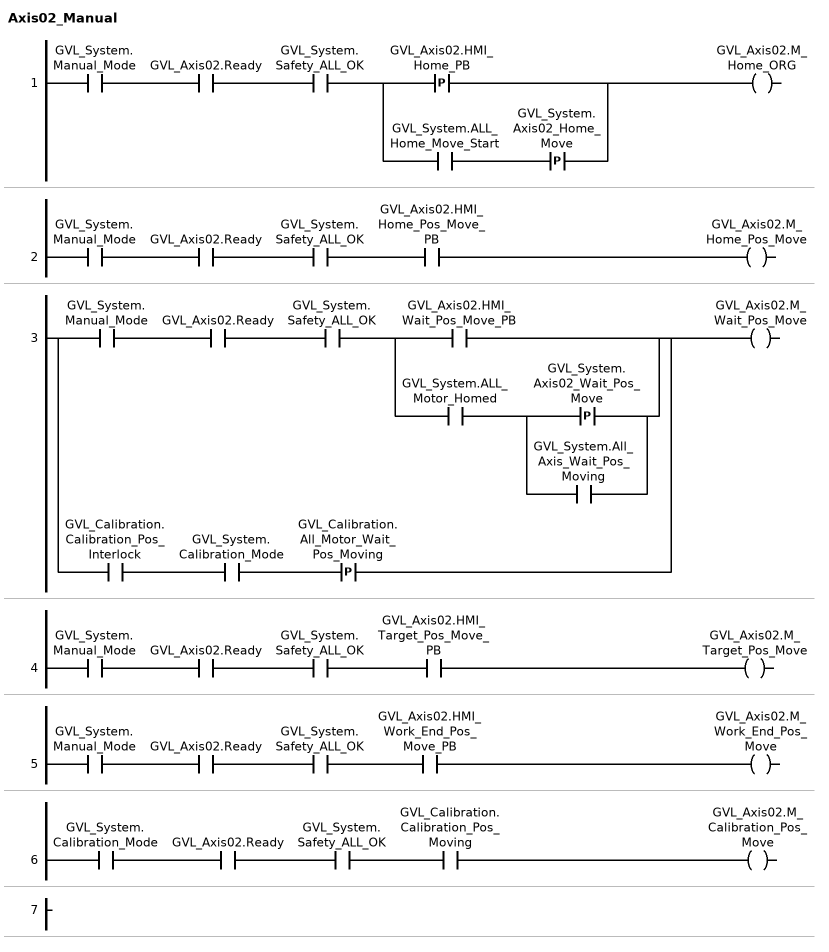
// NETWORK 1
_rt1(CLK := GVL_Axis02.HMI_Home_PB);
_rt2(CLK := GVL_System.Axis02_Home_Move);
GVL_Axis02.M_Home_ORG := GVL_System.Manual_Mode AND GVL_Axis02.Ready AND GVL_System.Safety_ALL_OK AND (_rt1.Q OR GVL_System.ALL_Home_Move_Start AND _rt2.Q);

// NETWORK 2
GVL_Axis02.M_Home_Pos_Move := GVL_System.Manual_Mode AND GVL_Axis02.Ready AND GVL_System.Safety_ALL_OK AND GVL_Axis02.HMI_Home_Pos_Move_PB;

// NETWORK 3
_rt3(CLK := GVL_System.Axis02_Wait_Pos_Move);
_rt4(CLK := GVL_Calibration.All_Motor_Wait_Pos_Moving);
GVL_Axis02.M_Wait_Pos_Move := GVL_System.Manual_Mode AND GVL_Axis02.Ready AND GVL_System.Safety_ALL_OK AND (GVL_Axis02.HMI_Wait_Pos_Move_PB OR GVL_System.ALL_Motor_Homed AND (_rt3.Q OR GVL_System.All_Axis_Wait_Pos_Moving)) OR GVL_Calibration.Calibration_Pos_Interlock AND GVL_System.Calibration_Mode AND _rt4.Q;

// NETWORK 4
GVL_Axis02.M_Target_Pos_Move := GVL_System.Manual_Mode AND GVL_Axis02.Ready AND GVL_System.Safety_ALL_OK AND GVL_Axis02.HMI_Target_Pos_Move_PB;

// NETWORK 5
GVL_Axis02.M_Work_End_Pos_Move := GVL_System.Manual_Mode AND GVL_Axis02.Ready AND GVL_System.Safety_ALL_OK AND GVL_Axis02.HMI_Work_End_Pos_Move_PB;

// NETWORK 6
GVL_Axis02.M_Calibration_Pos_Move := GVL_System.Calibration_Mode AND GVL_Axis02.Ready AND GVL_System.Safety_ALL_OK AND GVL_Calibration.Calibration_Pos_Moving;

// NETWORK 7

END_PROGRAM

// ---- POUs/Axis02_X/Axis02_Auto.TcPOU
PROGRAM Axis02_Auto
VAR
//System_Bit
	Always_ON	:	BOOL	:=TRUE	;//상시 ON 
	Always_OFF	:	BOOL	:=FALSE	;//상시 OFF
END_VAR

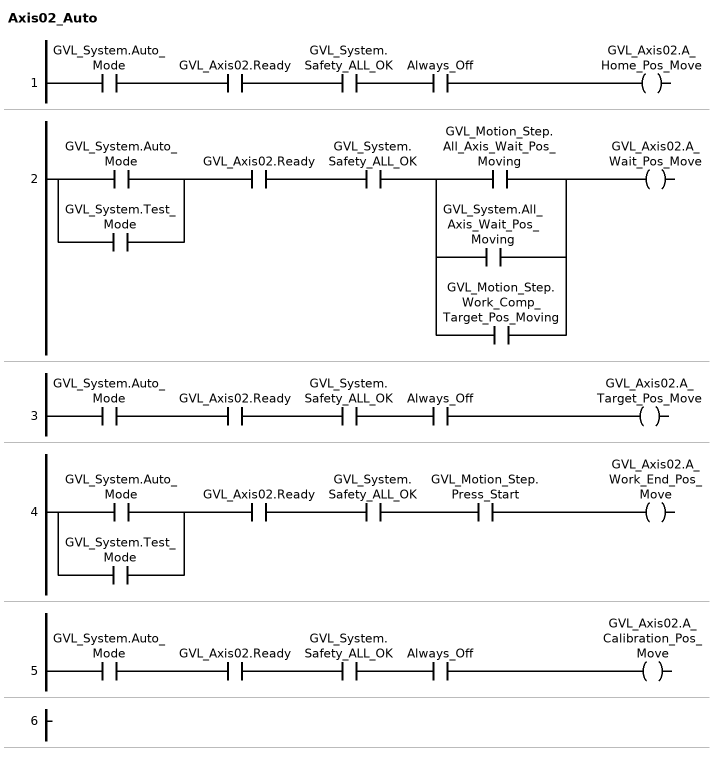
// NETWORK 1
GVL_Axis02.A_Home_Pos_Move := GVL_System.Auto_Mode AND GVL_Axis02.Ready AND GVL_System.Safety_ALL_OK AND Always_Off;

// NETWORK 2
GVL_Axis02.A_Wait_Pos_Move := (GVL_System.Auto_Mode OR GVL_System.Test_Mode) AND GVL_Axis02.Ready AND GVL_System.Safety_ALL_OK AND (GVL_Motion_Step.All_Axis_Wait_Pos_Moving OR GVL_System.All_Axis_Wait_Pos_Moving OR GVL_Motion_Step.Work_Comp_Target_Pos_Moving);

// NETWORK 3
GVL_Axis02.A_Target_Pos_Move := GVL_System.Auto_Mode AND GVL_Axis02.Ready AND GVL_System.Safety_ALL_OK AND Always_Off;

// NETWORK 4
GVL_Axis02.A_Work_End_Pos_Move := (GVL_System.Auto_Mode OR GVL_System.Test_Mode) AND GVL_Axis02.Ready AND GVL_System.Safety_ALL_OK AND GVL_Motion_Step.Press_Start;

// NETWORK 5
GVL_Axis02.A_Calibration_Pos_Move := GVL_System.Auto_Mode AND GVL_Axis02.Ready AND GVL_System.Safety_ALL_OK AND Always_Off;

// NETWORK 6

END_PROGRAM

// ---- POUs/Axis02_X/Axis02_Alarm.TcPOU
PROGRAM Axis02_Alarm
VAR
//System_Bit
	Always_ON	:	BOOL	:=TRUE	;//상시 ON 
	Always_OFF	:	BOOL	:=FALSE	;//상시 OFF
END_VAR

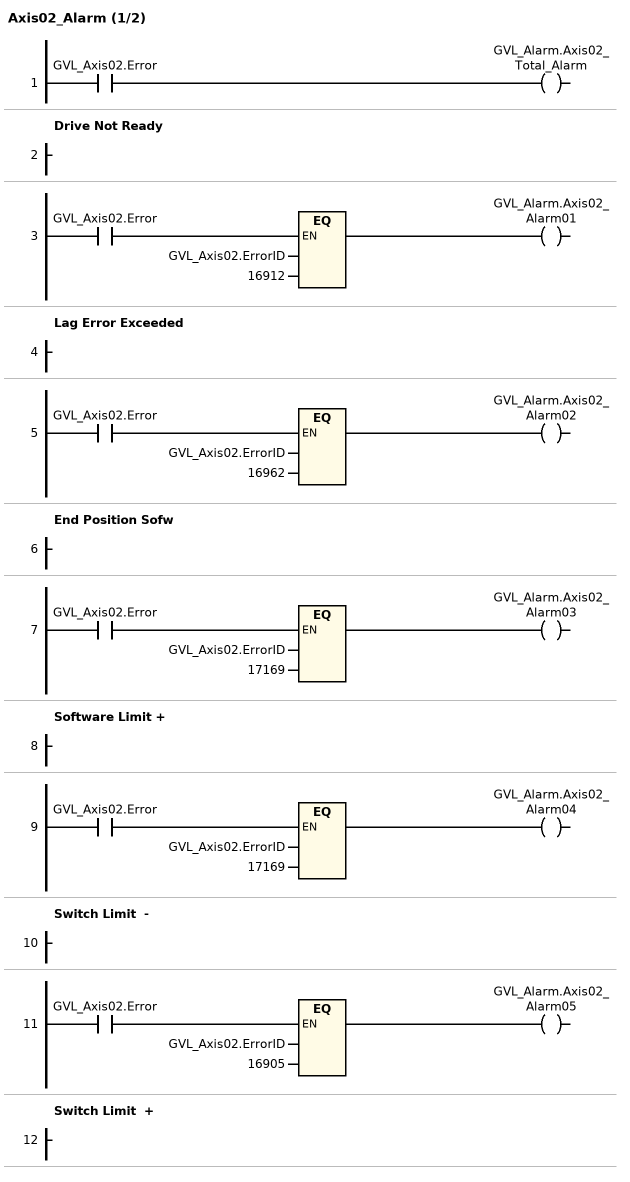
// NETWORK 1
GVL_Alarm.Axis02_Total_Alarm := GVL_Axis02.Error;

// NETWORK 2: Drive Not Ready

// NETWORK 3
GVL_Alarm.Axis02_Alarm01 := GVL_Axis02.Error AND GVL_Axis02.ErrorID = 16912;

// NETWORK 4: Lag Error Exceeded

// NETWORK 5
GVL_Alarm.Axis02_Alarm02 := GVL_Axis02.Error AND GVL_Axis02.ErrorID = 16962;

// NETWORK 6: End Position Sofw

// NETWORK 7
GVL_Alarm.Axis02_Alarm03 := GVL_Axis02.Error AND GVL_Axis02.ErrorID = 17169;

// NETWORK 8: Software Limit +

// NETWORK 9
GVL_Alarm.Axis02_Alarm04 := GVL_Axis02.Error AND GVL_Axis02.ErrorID = 17169;

// NETWORK 10: Switch Limit -

// NETWORK 11
GVL_Alarm.Axis02_Alarm05 := GVL_Axis02.Error AND GVL_Axis02.ErrorID = 16905;

// NETWORK 12: Switch Limit +

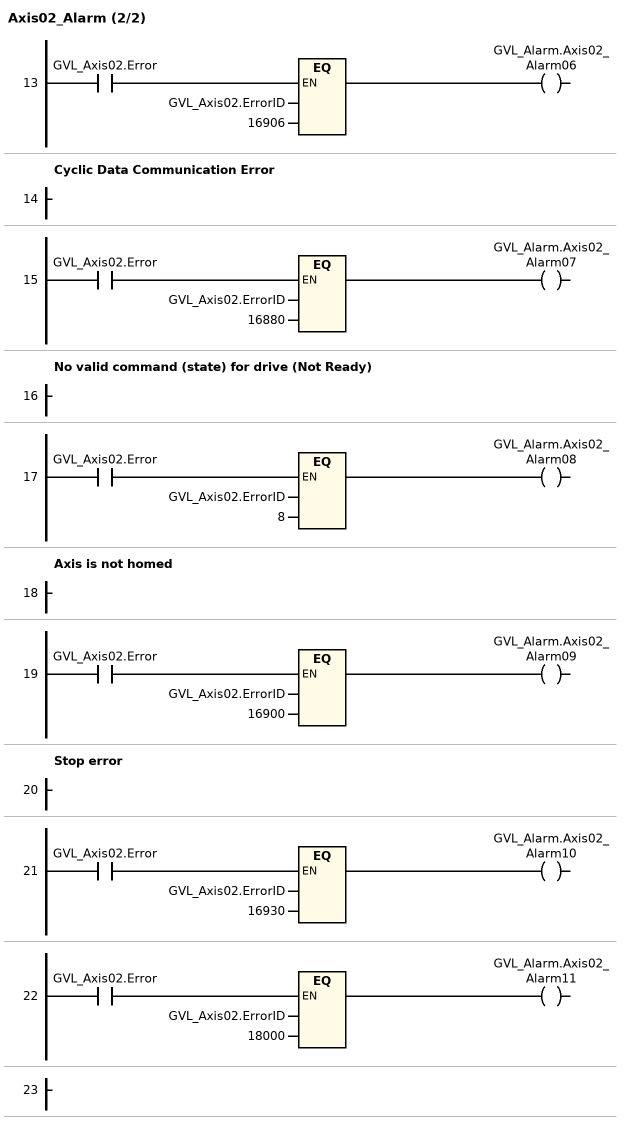
// NETWORK 13
GVL_Alarm.Axis02_Alarm06 := GVL_Axis02.Error AND GVL_Axis02.ErrorID = 16906;

// NETWORK 14: Cyclic Data Communication Error

// NETWORK 15
GVL_Alarm.Axis02_Alarm07 := GVL_Axis02.Error AND GVL_Axis02.ErrorID = 16880;

// NETWORK 16: No valid command (state) for drive (Not Ready)

// NETWORK 17
GVL_Alarm.Axis02_Alarm08 := GVL_Axis02.Error AND GVL_Axis02.ErrorID = 8;

// NETWORK 18: Axis is not homed

// NETWORK 19
GVL_Alarm.Axis02_Alarm09 := GVL_Axis02.Error AND GVL_Axis02.ErrorID = 16900;

// NETWORK 20: Stop error

// NETWORK 21
GVL_Alarm.Axis02_Alarm10 := GVL_Axis02.Error AND GVL_Axis02.ErrorID = 16930;

// NETWORK 22
GVL_Alarm.Axis02_Alarm11 := GVL_Axis02.Error AND GVL_Axis02.ErrorID = 18000;

// NETWORK 23

END_PROGRAM

// ---- POUs/Axis03_Y/Axis03_Status.TcPOU
PROGRAM Axis03_Status
VAR
//System_Bit
	Always_ON	:	BOOL	:=TRUE	;//상시 ON 
	Always_OFF	:	BOOL	:=FALSE	;//상시 OFF
	
//Motor_Command
	Axis03_Status_01: MC_ReadStatus;
	Axis03_Position_Read_01: MC_ReadActualPosition;
	Axis03_Velocity_Read_01: MC_ReadActualVelocity;
	Axis03_Reset_01: MC_Reset;
	Axis03_Stop_01: MC_Stop;
END_VAR

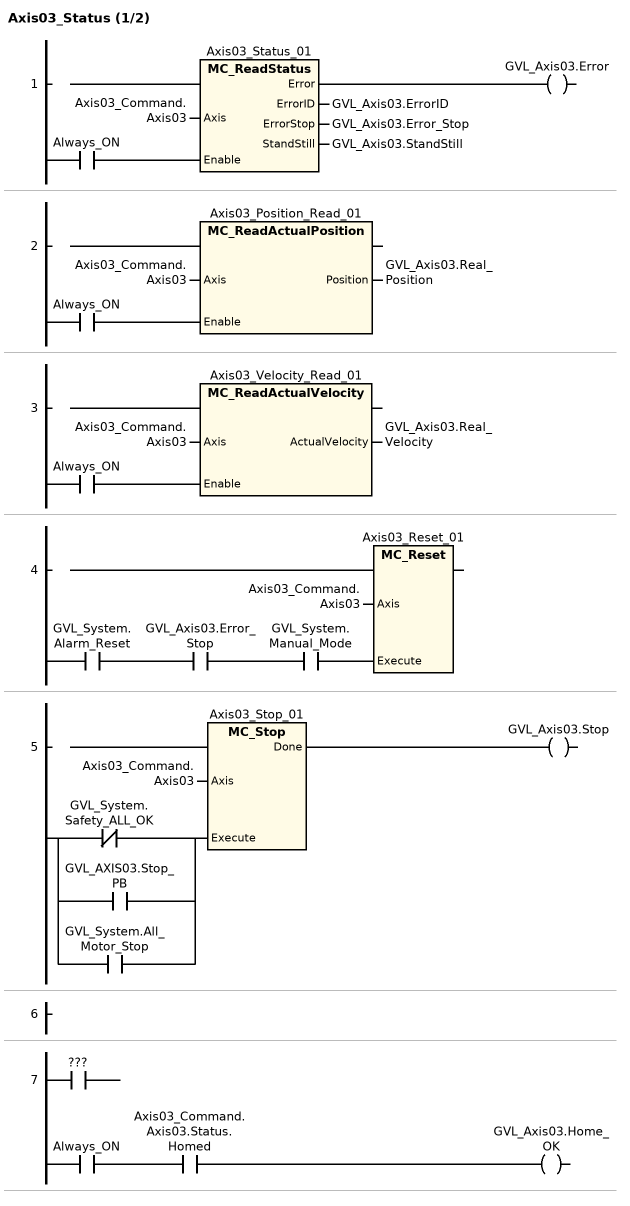
// NETWORK 1
Axis03_Status_01(
    Axis := Axis03_Command.Axis03,
    Enable := Always_ON,
    Error => GVL_Axis03.Error,
    ErrorID => GVL_Axis03.ErrorID,
    ErrorStop => GVL_Axis03.Error_Stop,
    StandStill => GVL_Axis03.StandStill); // MC_ReadStatus

// NETWORK 2
Axis03_Position_Read_01(
    Axis := Axis03_Command.Axis03,
    Enable := Always_ON,
    Position => GVL_Axis03.Real_Position); // MC_ReadActualPosition

// NETWORK 3
Axis03_Velocity_Read_01(
    Axis := Axis03_Command.Axis03,
    Enable := Always_ON,
    ActualVelocity => GVL_Axis03.Real_Velocity); // MC_ReadActualVelocity

// NETWORK 4
Axis03_Reset_01(Axis := Axis03_Command.Axis03, Execute := GVL_System.Alarm_Reset AND GVL_Axis03.Error_Stop AND GVL_System.Manual_Mode); // MC_Reset

// NETWORK 5
Axis03_Stop_01(Axis := Axis03_Command.Axis03, Execute := NOT GVL_System.Safety_ALL_OK OR GVL_AXIS03.Stop_PB OR GVL_System.All_Motor_Stop); // MC_Stop
GVL_Axis03.Stop := Axis03_Stop_01.Done;

// NETWORK 6

// NETWORK 7
GVL_Axis03.Home_OK := Always_ON AND Axis03_Command.Axis03.Status.Homed;

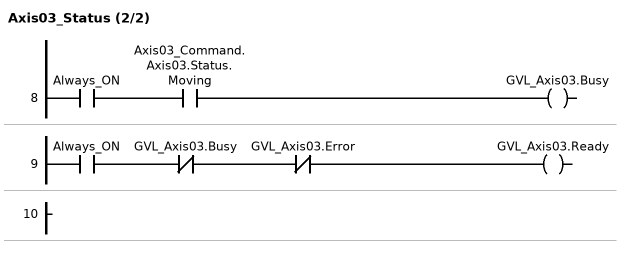
// NETWORK 8
GVL_Axis03.Busy := Always_ON AND Axis03_Command.Axis03.Status.Moving;

// NETWORK 9
GVL_Axis03.Ready := Always_ON AND NOT GVL_Axis03.Busy AND NOT GVL_Axis03.Error;

// NETWORK 10

END_PROGRAM

// ---- POUs/Axis03_Y/Axis03_Command.TcPOU
PROGRAM Axis03_Command
VAR
//System_Bit
	Always_ON	:	BOOL	:=TRUE	;//상시 ON 
	Always_OFF	:	BOOL	:=FALSE	;//상시 OFF

//Motor_Command
	Axis03: AXIS_REF;											//Y축
	Axis03_MC_Power: MC_Power;
	Axis03_MC_Home: FB_HomeBeforeMoveAX8000;
	Axis03_Jog: MC_Jog;	
	Axis03_Home_Pos_Move: MC_MoveAbsolute;
	Axis03_Wait_Pos_Move: MC_MoveAbsolute;
	Axis03_Target_Pos_Move: MC_MoveAbsolute;
	Axis03_Work_End_Move: MC_MoveAbsolute;
	Axis03_Maint_Move: MC_MoveAbsolute;
	Axis03_Tool_Change: MC_MoveAbsolute;	
	Axis03_Calibration: MC_MoveAbsolute;	

	Timer02: TON;
	keb_Y: BOOL;
	Axis03_ku_Pos_Move: MC_MoveAbsolute;
	keb_Y_data_PB: BOOL;
END_VAR
VAR // added by the converter: edge detectors and wires of the graphical bodies
    _rt1, _rt2, _rt3 : R_TRIG;
END_VAR

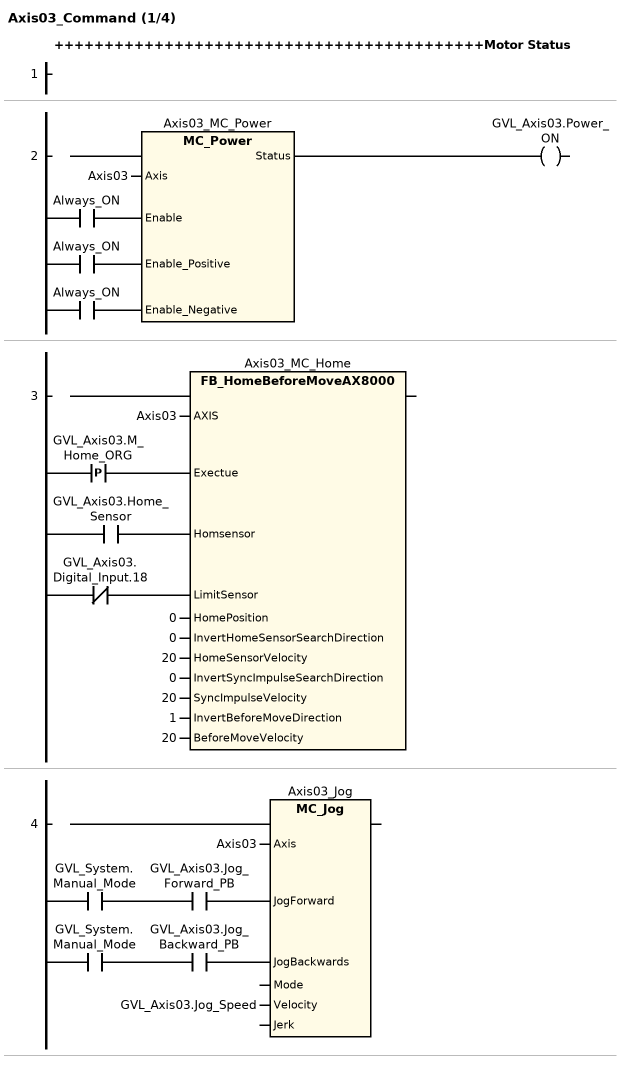
// NETWORK 1: +++++++++++++++++++++++++++++++++++++++++++Motor Status

// NETWORK 2
Axis03_MC_Power(
    Axis := Axis03,
    Enable := Always_ON,
    Enable_Positive := Always_ON,
    Enable_Negative := Always_ON); // MC_Power
GVL_Axis03.Power_ON := Axis03_MC_Power.Status;

// NETWORK 3
_rt1(CLK := GVL_Axis03.M_Home_ORG);
Axis03_MC_Home(
    AXIS := Axis03,
    Exectue := _rt1.Q,
    Homsensor := GVL_Axis03.Home_Sensor,
    LimitSensor := NOT GVL_Axis03.Digital_Input.18,
    HomePosition := 0,
    InvertHomeSensorSearchDirection := 0,
    HomeSensorVelocity := 20,
    InvertSyncImpulseSearchDirection := 0,
    SyncImpulseVelocity := 20,
    InvertBeforeMoveDirection := 1,
    BeforeMoveVelocity := 20); // FB_HomeBeforeMoveAX8000

// NETWORK 4
Axis03_Jog(
    Axis := Axis03,
    JogForward := GVL_System.Manual_Mode AND GVL_Axis03.Jog_Forward_PB,
    JogBackwards := GVL_System.Manual_Mode AND GVL_Axis03.Jog_Backward_PB,
    Velocity := GVL_Axis03.Jog_Speed); // MC_Jog

